		IF ((phase_horizontal_slave_position > (csp_case_feed_shuttle_horizontal.axis.actual_position + 5))
			OR
			(phase_horizontal_slave_position < (csp_case_feed_shuttle_horizontal.axis.actual_position - 5)))
		THEN
			large_move_required := TRUE;	// shuttle is moving a large amount, spreader need to be moved
		ELSE
			large_move_required := FALSE; // shuttle is moving a small amount, spreaders do not need to be moved
		END_IF
		
		IF (ABSENT_HOR_VER = FALSE) 
			AND (csp_case_flapControl.spreaders_clear
			OR
			large_move_required = FALSE)
		THEN
			axis_move_absolute(
				position 		:= phase_horizontal_slave_position,
				velocity 		:= csp_case_feed_shuttle_horizontal.MOTOR_PHASE_VELOCITY_MMPS,
				direction		:= AXIS_CURRENT_DIRECTION,
				acceleration 	:= csp_case_feed_shuttle_horizontal.MOTOR_MAX_ACCELLERATION_MMPS2,
				deceleration 	:= csp_case_feed_shuttle_horizontal.MOTOR_MAX_DECELLERATION_MMPS2, 
				jerk 			:=csp_case_feed_shuttle_horizontal. MOTOR_MAX_JERK_MMPS3, 
				buffer_mode 	:= AXIS_BUFFER_MODE_BUFFERED,
				CONVERSION_this := csp_case_feed_shuttle_horizontal.axis); 
	
			axis_move_absolute(
				position 		:= phase_vertical_slave_position,
				velocity 		:= csp_case_feed_shuttle_vertical.MOTOR_PHASE_VELOCITY_DEGPS,
				direction		:= AXIS_SHORTEST_WAY,
				acceleration 	:= csp_case_feed_shuttle_vertical.MOTOR_MAX_ACCELLERATION_DEGPS2,
				deceleration 	:= csp_case_feed_shuttle_vertical.MOTOR_MAX_DECELLERATION_DEGPS2, 
				jerk 			:= csp_case_feed_shuttle_vertical.MOTOR_MAX_JERK_DEGPS3, 
				buffer_mode 	:= AXIS_BUFFER_MODE_BUFFERED,
				CONVERSION_this := csp_case_feed_shuttle_vertical.axis); 
		END_IF
	 	
	
			axis_move_absolute(
				position 		:= phase_x_slave_position,
				velocity 		:= csp_case_feed_kinematic_x.MOTOR_PHASE_VELOCITY_MMPS,
				direction		:= AXIS_CURRENT_DIRECTION,
				acceleration 	:= csp_case_feed_kinematic_x.MOTOR_MAX_ACCELLERATION_MMPS2,
				deceleration 	:= csp_case_feed_kinematic_x.MOTOR_MAX_DECELLERATION_MMPS2, 
				jerk 			:= csp_case_feed_kinematic_x.MOTOR_MAX_JERK_MMPS3, 
				buffer_mode 	:= AXIS_BUFFER_MODE_BUFFERED,
				CONVERSION_this := csp_case_feed_kinematic_x.axis); 
			
			axis_move_absolute(
				position 		:= phase_y_slave_position,
				velocity 		:= csp_case_feed_kinematic_y.MOTOR_PHASE_VELOCITY_MMPS,
				direction		:= AXIS_CURRENT_DIRECTION,
				acceleration 	:= csp_case_feed_kinematic_y.MOTOR_MAX_ACCELLERATION_MMPS2,
				deceleration 	:= csp_case_feed_kinematic_y.MOTOR_MAX_DECELLERATION_MMPS2, 
				jerk 			:= csp_case_feed_kinematic_y.MOTOR_MAX_JERK_MMPS3, 
				buffer_mode 	:= AXIS_BUFFER_MODE_BUFFERED,
				CONVERSION_this := csp_case_feed_kinematic_y.axis); 
			
			axis_move_absolute(
				position 		:= phase_tilt_slave_position,
				velocity 		:= csp_case_feed_kinematic_tilt.MOTOR_PHASE_VELOCITY_DEGPS,
				direction		:= AXIS_CURRENT_DIRECTION,
				acceleration 	:= csp_case_feed_kinematic_tilt.MOTOR_MAX_ACCELLERATION_DEGPS2,
				deceleration 	:= csp_case_feed_kinematic_tilt.MOTOR_MAX_DECELLERATION_DEGPS2, 
				jerk 			:= csp_case_feed_kinematic_tilt.MOTOR_MAX_JERK_DEGPS3, 
				buffer_mode 	:= AXIS_BUFFER_MODE_BUFFERED,
				CONVERSION_this := csp_case_feed_kinematic_tilt.axis); 
			
		IF 	axis_is_absolute_moving(csp_case_feed_shuttle_horizontal.axis)
			AND
			axis_is_absolute_moving(csp_case_feed_shuttle_vertical.axis)
			AND
			axis_is_absolute_moving(csp_case_feed_kinematic_x.axis)
			AND
			axis_is_absolute_moving(csp_case_feed_kinematic_y.axis)
			AND
			axis_is_absolute_moving(csp_case_feed_kinematic_tilt.axis)
		THEN
			csp_case_feed_kinematic.ext_phase_request := TRUE;
			phase_status_next := CSP_CASE_FEED_STATUS_PHASE_MOVED_SLAVE_POSITION;
		ELSIF 	ABSENT_HOR_VER
				AND
				axis_is_absolute_moving(csp_case_feed_kinematic_x.axis)
				AND
				axis_is_absolute_moving(csp_case_feed_kinematic_y.axis)
				AND
				axis_is_absolute_moving(csp_case_feed_kinematic_tilt.axis)
		THEN
				csp_case_feed_kinematic.ext_phase_request := TRUE;
				phase_status_next := CSP_CASE_FEED_STATUS_PHASE_MOVED_SLAVE_POSITION;
		END_IF

		
	CSP_CASE_FEED_STATUS_PHASE_MOVED_SLAVE_POSITION:
	
		IF 	((axis_is_standstill(csp_case_feed_shuttle_horizontal.axis)
			AND
			axis_is_standstill(csp_case_feed_shuttle_vertical.axis))
			OR
			ABSENT_HOR_VER)
			AND
			axis_is_standstill(csp_case_feed_kinematic_x.axis)
			AND
			axis_is_standstill(csp_case_feed_kinematic_y.axis)
			AND
			axis_is_standstill(csp_case_feed_kinematic_tilt.axis)
			AND
			csp_case_feed_kinematic.phase_request
		THEN			
			phase_status_next := CSP_CASE_FEED_STATUS_PHASE_DONE;
		END_IF
					
		
	CSP_CASE_FEED_STATUS_PHASE_DONE:	(* Phase done *)
			
		phase_running := FALSE;
		phase_done := TRUE;			

		IF 	csp_case_feed_kinematic.ext_stop_request	
		THEN
			phase_done := FALSE;
			phase_status_next := CSP_CASE_FEED_STATUS_PHASE_START;
		END_IF
		
		
	CSP_CASE_FEED_STATUS_PHASE_ERROR:	(* Phase error *)
	
		IF	phase_running
		THEN
			axis_disable(csp_case_feed_shuttle_horizontal.axis);
			axis_disable(csp_case_feed_shuttle_vertical.axis);									
		END_IF
		phase_running := FALSE;
		
		IF	phase_conditions 	
		THEN
			phase_status_next := CSP_CASE_FEED_STATUS_PHASE_START;
		END_IF
		
END_CASE

IF 	NOT debug_state_machine
	OR
	debug_phase_machine_one_step	
THEN
	phase_status := phase_status_next;
	debug_phase_machine_one_step := FALSE;
END_IF

(* Phasing timeout *)
IF	phase_running
	AND NOT debug_state_machine
THEN
	IF	timer_is_expired(phase_time_out_tmr)
	THEN
		process_message_set(1, phase_status, 0, phase_faulted_aem);
	END_IF
ELSE
	timer_restart(30000, phase_time_out_tmr);
END_IF
END_ACTION

END_PROGRAM

// ---- POUs/AFL extensions/jog_manager/status/jog_manager_is_jog_axis_active.TcPOU
(*$
	Returns <i>TRUE</i> if the status of the instance <b><i>this</i></b> is
	<a href="#jog_manager_status_enum"><i>JOG_MANAGER_STATUS_ACTIVE</i></a>
	and  <i>list_selected</i> is a valid index,
	<i>FALSE</i> otherwise.
$*)
FUNCTION jog_manager_is_jog_axis_active : BOOL
VAR_INPUT
	index:				UINT;
END_VAR
VAR_IN_OUT
    CONVERSION_this:	jog_manager;	(*$ Instance to which the method applies $*)
END_VAR

IF	(
		(CONVERSION_this.CONVERSION_private.list_selected = index)
		OR 	
		(CONVERSION_this.CONVERSION_private.old_list_selected = index)
	)
	AND
	CONVERSION_this.CONVERSION_private.list_selected_axis_is_valid
THEN
	jog_manager_is_jog_axis_active := (CONVERSION_this.status >= JOG_MANAGER_STATUS_ACTIVE);
ELSE
	jog_manager_is_jog_axis_active := FALSE;
END_IF

END_FUNCTION

// ---- Application/CSP/Case/Feed/Kinematic/csp_case_feed_kinematic.TcPOU
(*********************************** G.D S.p.A. - Technical Department ***********************************
============= PROGRAM INFO ============
FOLDER:             TBD
MACHINES INVOLVED:  TBD 

============= DESCRIPTION =============
csp machine declaration

============= REVISIONS ===============
Date		Version	 	Author      	Description             
----------	-------		------------  	--------------------------------------------
2019/04/05 	0000.00	 	M.Grasso		Creation of the PRG

**********************************************************************************************************)
(*$R process_ref := prc; $*)
PROGRAM csp_case_feed_kinematic
VAR_INPUT
	ext_cartesian_mode_request:						BOOL;
	ext_phase_request:								BOOL;
	ext_stop_request:								BOOL;
END_VAR
VAR
	
	prc:											process;
	prc_path:										STRING;
	
	in_stKinToPlc	AT %I*:							NcToPlc_NciChannel_Ref;
	out_stPlcToKin	AT %Q*:							PlcTonc_NciChannel_Ref;
	stAxesConfig:									ST_KinAxes;
	stAxesPosIn:									ARRAY[1..8] OF LREAL;
	stAxesPosOut:									ARRAY[1..8] OF LREAL;
	uMetaInfoIn:									U_KinMetaInfo;
	uMetaInfoOut:									U_KinMetaInfo;
		
	kin_config_execute:								BOOL := FALSE;
	kin_config_cartesian_mode:						BOOL := FALSE;
	fbConfigKinGroup:								FB_KinConfigGroup;
	kin_config_group_aem:	 						message;	
	kin_cacl_execute:								BOOL := FALSE;
	fbCalcKinTrafo:									FB_KinCalcTRafo;
	fbResetKinGroup:								FB_KinResetGroup;
	
	fsm_enable_condition:							BOOL := FALSE;
	fsm_next_status:								csp_case_feed_kinematic_status_enum;
	fsm_status:										csp_case_feed_kinematic_status_enum;
			
	kinematic_jog_on:								BOOL := FALSE; (*$P $*)
	kinematic_jog_on_motcond:						motorization_conditioner;
	
	memo_cartesian_mode_request:					BOOL;
	memo_phase_request:								BOOL;
	memo_stop_request:								BOOL;
	
	cartesian_mode_active:							BOOL;
	is_ok:											BOOL;
	is_axis_enabled:								BOOL;
	
	disable_req:									BOOL := FALSE;
	move_kinematic:									BOOL := TRUE;
	enable_kinematic:								BOOL := TRUE;
	engage_enable:									BOOL := FALSE;
	disable_kinematic:								BOOL := TRUE;
	
	//Cmd	
	joint_cartesian_mode:							BOOL := FALSE;
	join_cartesian_mode_RTRIG:						R_TRIG;
	
	elbow_jog_plus:									BOOL := FALSE;
	elbow_jog_minus:								BOOL := FALSE;
	elbow_phase_move:								BOOL := FALSE;
	elbow_copy_phase:								BOOL := FALSE;
	
	shoulder_jog_plus:								BOOL := FALSE;
	shoulder_jog_minus:								BOOL := FALSE;
	shoulder_phase_move:							BOOL := FALSE;
	shoulder_copy_phase:							BOOL := FALSE;
	
	wrist_jog_plus:									BOOL := FALSE;
	wrist_jog_minus:								BOOL := FALSE;
	wrist_phase_move:								BOOL := FALSE;	
	wrist_copy_phase:								BOOL := FALSE;	

	x_jog_plus:										BOOL := FALSE;
	x_jog_minus:									BOOL := FALSE;
	x_phase_move:									BOOL := FALSE;
	x_copy_phase:									BOOL := FALSE;
	
	y_jog_plus:										BOOL := FALSE;
	y_jog_minus:									BOOL := FALSE;
	y_phase_move:									BOOL := FALSE;
	y_copy_phase:									BOOL := FALSE;
	
	tilt_jog_plus:									BOOL := FALSE;
	tilt_jog_minus:									BOOL := FALSE;
	tilt_phase_move:								BOOL := FALSE;	
	tilt_copy_phase:								BOOL := FALSE;
	
	elbow_move_speed:								LREAL := 5.0; 		(*$P unit := °/s; $*)
	shoulder_move_speed:							LREAL := 5.0;		(*$P unit := °/s; $*)
	wrist_move_speed:								LREAL := 5.0;		(*$P unit := °/s; $*)
	x_move_speed:									LREAL := 10.0;		(*$P unit := mm/s; $*)
	y_move_speed:									LREAL := 10.0;		(*$P unit := mm/s; $*)
	tilt_move_speed:								LREAL := 10.0;		(*$P unit := °/s; $*)
	
	phase_move_speed:								LREAL := 10;
	phase_move_time:								LREAL;
	x_phase_distance:								LREAL;
	x_phase_move_speed:								LREAL;
	y_phase_distance:								LREAL;	
	y_phase_move_speed:								LREAL;	
		
	phase_request:									BOOL := FALSE;
	elbow_phase_position:							LREAL := 0.0;		(*$P step := 0.001; unit := °; $*)
	elbow_phase_position_pow:						parameter_overwrite;
	shoulder_phase_position:						LREAL := 45.0;		(*$P step := 0.001; unit := °; $*)
	shoulder_phase_position_pow:					parameter_overwrite;
	wrist_phase_position:							LREAL := 0.0;		(*$P step := 0.001; unit := °; $*)
	wrist_phase_position_pow:						parameter_overwrite;
	x_phase_position:								LREAL := -554;		(*$P step := 0.001; unit := mm; $*)
	x_phase_position_pow:							parameter_overwrite;
	y_phase_position:								LREAL := -660.3;	(*$P step := 0.001; unit := mm; $*)
	y_phase_position_pow:							parameter_overwrite;
	tilt_phase_position:							LREAL := 45.0;		(*$P step := 0.001; unit := °; $*)
	tilt_phase_position_pow:						parameter_overwrite;
	
	elbow_actual_position:							LREAL;				(*$M step := 0.001; unit := °; $*)
	shoulder_actual_position:						LREAL;				(*$M step := 0.001; unit := °; $*)
	wrist_actual_position:							LREAL;				(*$M step := 0.001; unit := °; $*)
	x_actual_position:								LREAL;				(*$M step := 0.01; unit := mm; $*)
	y_actual_position:								LREAL;				(*$M step := 0.01; unit := mm; $*)
	tilt_actual_position:							LREAL;				(*$M step := 0.01; unit := °; $*)
	axis_are_moving:								BOOL;
	axis_are_phase_moving:							BOOL;
	
	//Visu variable management	
	visu_disable_general_command:					BOOL;
	visu_disable_ACS_command:						BOOL;
	visu_disable_MCS_command:						BOOL;
	visu_disable_ACS_jog_mode:						BOOL;
	visu_disable_MCS_jog_mode:						BOOL;
	visu_disable_phase_request:						BOOL;
	
	//HMI custom page variable management
	hmi_joint_cartesian_mode_cbtn:					command_button;
	hmi_phase_request_cbtn:							command_button;
	hmi_phase_request_cbtn_is_pressed:				BOOL;	
	
	hmi_elbow_jog_plus_cbtn:						command_button;
	hmi_elbow_jog_minus_cbtn:						command_button;
	hmi_elbow_phase_move_cbtn:						command_button;
	hmi_elbow_copy_phase_cbtn:						command_button;
	hmi_elbow_activate_pendant_cbtn:				command_button;
	hmi_elbow_activate_pendant_cbtn_is_pressed:		BOOL;
	hmi_elbow_pendant_active:						BOOL := FALSE;
	
	hmi_shoulder_jog_plus_cbtn:						command_button;
	hmi_shoulder_jog_minus_cbtn:					command_button;
	hmi_shoulder_phase_move_cbtn:					command_button;
	hmi_shoulder_copy_phase_cbtn:					command_button;
	hmi_shoulder_activate_pendant_cbtn:				command_button;
	hmi_shoulder_activate_pendant_cbtn_is_pressed:	BOOL;
	hmi_shoulder_pendant_active:					BOOL := FALSE;
	
	hmi_wrist_jog_plus_cbtn:						command_button;
	hmi_wrist_jog_minus_cbtn:						command_button;
	hmi_wrist_phase_move_cbtn:						command_button;
	hmi_wrist_copy_phase_cbtn:						command_button;
	hmi_wrist_activate_pendant_cbtn:				command_button;
	hmi_wrist_activate_pendant_cbtn_is_pressed:		BOOL;
	hmi_wrist_pendant_active:						BOOL := FALSE;
	
	hmi_x_jog_plus_cbtn:							command_button;
	hmi_x_jog_minus_cbtn:							command_button;
	hmi_x_phase_move_cbtn:							command_button;
	hmi_x_copy_phase_cbtn:							command_button;
	hmi_x_activate_pendant_cbtn:					command_button;
	hmi_x_activate_pendant_cbtn_is_pressed:			BOOL;
	hmi_x_pendant_active:							BOOL := FALSE;
	
	hmi_y_jog_plus_cbtn:							command_button;
	hmi_y_jog_minus_cbtn:							command_button;
	hmi_y_phase_move_cbtn:							command_button;
	hmi_y_copy_phase_cbtn:							command_button;
	hmi_y_activate_pendant_cbtn:					command_button;
	hmi_y_activate_pendant_cbtn_is_pressed:			BOOL;
	hmi_y_pendant_active:							BOOL := FALSE;
	
	hmi_tilt_jog_plus_cbtn:							command_button;
	hmi_tilt_jog_minus_cbtn:						command_button;
	hmi_tilt_phase_move_cbtn:						command_button;
	hmi_tilt_copy_phase_cbtn:						command_button;
	hmi_tilt_activate_pendant_cbtn:					command_button;
	hmi_tilt_activate_pendant_cbtn_is_pressed:		BOOL;
	hmi_tilt_pendant_active:						BOOL := FALSE;
	
	hmi_pendant_active:								BOOL;
	
	hmi_enable_general_command_hgos:				hmi_graphic_object_status;
	hmi_enable_joint_hgos:							hmi_graphic_object_status;
	hmi_enable_cartesian_hgos:						hmi_graphic_object_status;
	hmi_enable_ACS_command_hgos:					hmi_graphic_object_status;
	hmi_enable_MCS_command_hgos:					hmi_graphic_object_status;
	hmi_enable_ACS_jog_mode_hgos:					hmi_graphic_object_status;
	hmi_enable_MCS_jog_mode_hgos:					hmi_graphic_object_status;
	hmi_enable_phase_request_hgos:					hmi_graphic_object_status;
	
	debug_phase_elbow:								BOOL := FALSE;
	debug_phase_shoulder:							BOOL := FALSE;
	debug_phase_wrist:								BOOL := FALSE;
	debug_state_machine:							BOOL := FALSE;
	debug_state_machine_one_step:					BOOL := FALSE;
	
	master_scaling_deg:								LREAL := 1.0;
	x_scaling_mm:									LREAL := 1.0;
	x_old_scaling_mm:								LREAL := 1.0;
	y_scaling_mm:									LREAL := 1.0;
	y_old_scaling_mm:								LREAL := 1.0;
	tilt_scaling_deg:								LREAL := 1.0;
	tilt_old_scaling_deg:							LREAL := 1.0;		
	Kinematic_tilt_error_aem: 						message;
	Kinematic_tilt_clear_error:						BOOL:= FALSE;
END_VAR

VAR CONSTANT	
	CONSTANTS:										csp_case_feed_kinematic_constant_struct;
	COIDTRAFO:										UDINT := 16#01010030;
END_VAR

_read_var_input();

_object_manager();

IF NOT objects_running()
THEN
	RETURN;	
END_IF

_read_process_image();

_mode_manager();

CASE process_get_mode(prc) of
	MODE_ABSENT,
	MODE_INACTIVE:
		RETURN;
	MODE_TEST:
		_handle_process_test();
END_CASE

_set_runtime_properties();

_hmi_Management();

(********************************* BODY *********************************)
(* Kinematic trasformation		
X		->		Shoulder (M1)
Y		->		Elbow (M2)			
Tilt	->		Wrist (M3)																											
*)	

stAxesConfig.nAxisIdsAcs[1] := csp_case_feed_arm_shoulder.axis.ax_ref.NcToPlc.AxisId; 
stAxesConfig.nAxisIdsAcs[2] := csp_case_feed_arm_elbow.axis.ax_ref.NcToPlc.AxisId;
stAxesConfig.nAxisIdsAcs[3] := csp_case_feed_arm_wrist.axis.ax_ref.NcToPlc.AxisId;

stAxesConfig.nAxisIdsMcs[1] := csp_case_feed_kinematic_x.axis.ax_ref.NcToPlc.AxisId;
stAxesConfig.nAxisIdsMcs[2] := csp_case_feed_kinematic_y.axis.ax_ref.NcToPlc.AxisId;
stAxesConfig.nAxisIdsMcs[3] := csp_case_feed_kinematic_tilt.axis.ax_ref.NcToPlc.AxisId;

fbConfigKinGroup(
	bExecute		:= kin_config_execute
					   OR
					   (
						   (
							   NOT axis_is_ok(FALSE, csp_case_feed_arm_elbow.axis)
							   OR
							   NOT axis_is_ok(FALSE, csp_case_feed_arm_shoulder.axis)
							   OR
							   NOT axis_is_ok(FALSE, csp_case_feed_arm_wrist.axis)	
							   OR
							   fbConfigKinGroup.bError
							)
							AND
 							csp_main.o_reset_button
					   ),
	bCartesianMode	:= kin_config_cartesian_mode, 
	stAxesList		:= stAxesConfig, 
	stKinRefIn		:= in_stKinToPlc, 
	bBusy			=> , 
	bDone			=> , 
	bError			=> , 
	nErrorId		=> );
	
fbResetKinGroup(
	bExecute		:= csp_main.o_reset_button
					AND 
					(in_stKinToPlc.ErrorCode <> 0), 
	nItpChannelId	:= 0, 
	stKinRefIn		:= in_stKinToPlc, 
	stAxesList		:= stAxesConfig, 
	bBusy			=> , 
	bDone			=> , 
	bError			=> , 
	nErrorId		=> );
	
kin_cacl_execute :=	NOT cartesian_mode_active
					AND
					NOT fbCalcKinTrafo.bBusy;
stAxesPosIn[1] := axis_get_actual_incremental_position(csp_case_feed_arm_shoulder.axis);
stAxesPosIn[2] := axis_get_actual_incremental_position(csp_case_feed_arm_elbow.axis);
stAxesPosIn[3] := axis_get_actual_incremental_position(csp_case_feed_arm_wrist.axis);
fbCalcKinTrafo(
	bExecute 		:= kin_cacl_execute,
	bForward 		:= NOT kin_config_cartesian_mode,
	oidTrafo 		:= COIDTRAFO,
	stAxesPosIn 	:= stAxesPosIn,
	stAxesPosOut 	:= stAxesPosOut,
	uMetaInfoIn		:= uMetaInfoIn ,
	uMetaInfoOut	:= uMetaInfoOut,
	bBusy			=> ,
	bDone			=> ,
	bError			=> ,
	nErrorId		=> );

(*Status*)
cartesian_mode_active := 
	(in_stKinToPlc.ChnOperationState = 4);
	
is_axis_enabled := (fsm_status = CSP_CASE_FEED_KINEMATIC_STATUS_ENABLED);
	

(* ALLOWS MACHINE TO RUN BECAUSE KINEMATIC IS NOT ON *)
IF motorization_manager_is_starting(csp_main_motorization_manager.motm)
AND NOT kinematic_jog_on
	THEN
		motorization_conditioner_start_done(kinematic_jog_on_motcond);
END_IF 


(*FSM Control*)
is_ok := 
	process_is_ready(prc)
	AND
	process_subtree_is_ready(prc)
	AND
	csp_case_feed_arm_elbow.servo_on_condition
	AND
	csp_case_feed_arm_shoulder.servo_on_condition
	AND
	csp_case_feed_arm_wrist.servo_on_condition
	AND
	axis_is_ok(FALSE, csp_case_feed_arm_elbow.axis)
	AND
	axis_is_ok(FALSE, csp_case_feed_arm_shoulder.axis)
	AND
	axis_is_ok(FALSE, csp_case_feed_arm_wrist.axis)						
	AND						
	axis_is_ok(FALSE, csp_case_feed_kinematic_x.axis)	
	AND
	axis_is_ok(FALSE, csp_case_feed_kinematic_y.axis)	
	AND
	axis_is_ok(FALSE, csp_case_feed_kinematic_tilt.axis)	
	AND												
	NOT fbConfigKinGroup.bError						
	AND
	NOT disable_req;
fsm_enable_condition := 
	is_ok
	AND
	(
		csp_case_feed_virtualMaster.is_ok
		OR
		(
			csp_main_accuChange.machine_size_running
			AND
			(
				NOT csp_case_feed_kinematic_x.in_accu_safe_pos
				OR
				NOT csp_case_feed_kinematic_y.in_accu_safe_pos
				OR
				NOT csp_case_feed_kinematic_tilt.in_accu_safe_pos
			)
		)
	);
	
IF	(
		NOT fsm_enable_condition
		OR
		(
			ext_stop_request 
			AND 
			NOT memo_stop_request
		)
	)
	AND
	fsm_status <> CSP_CASE_FEED_KINEMATIC_STATUS_DISABLED
	AND
	fsm_status < CSP_CASE_FEED_KINEMATIC_STATUS_STOP_REQUEST
THEN
	fsm_status	:=	CSP_CASE_FEED_KINEMATIC_STATUS_DISABLE_REQUEST;
	IF	ext_stop_request
	THEN
		fsm_next_status := fsm_status;
	END_IF
	phase_request:=FALSE;
END_IF

IF tilt_actual_position < 1200
	AND tilt_actual_position > 0
	AND csp_case_feed_kinematic_tilt.axis.actual_position < 1200   
	AND NOT Kinematic_tilt_clear_error
THEN
	process_message_set(1, 1, 1, Kinematic_tilt_error_aem);
ELSE
	process_message_reset(Kinematic_tilt_error_aem);
END_IF

IF process_message_is_on(Kinematic_tilt_error_aem)
	AND machine_is_stopped(csp.mch)
	OR machine_is_stop_emergency_active(csp.mch)
THEN
	process_message_reset(Kinematic_tilt_error_aem);
END_IF

CASE fsm_status OF
	
	CSP_CASE_FEED_KINEMATIC_STATUS_NOT_INITIALIZED:
	
        IF	axis_is_ok(return_when_absent := FALSE, CONVERSION_this := csp_case_feed_arm_elbow.axis)
			AND
			axis_is_ok(return_when_absent := FALSE, CONVERSION_this := csp_case_feed_arm_shoulder.axis)
			AND
			axis_is_ok(return_when_absent := FALSE, CONVERSION_this := csp_case_feed_arm_wrist.axis)
			AND
			axis_is_ok(return_when_absent := FALSE, CONVERSION_this := csp_case_feed_kinematic_x.axis)
			AND
			axis_is_ok(return_when_absent := FALSE, CONVERSION_this := csp_case_feed_kinematic_y.axis)
			AND
			axis_is_ok(return_when_absent := FALSE, CONVERSION_this := csp_case_feed_kinematic_tilt.axis)
        THEN
            fsm_next_status := CSP_CASE_FEED_KINEMATIC_STATUS_DISABLED;
        END_IF

		
	CSP_CASE_FEED_KINEMATIC_STATUS_DISABLED:
		
		IF	fsm_enable_condition
			AND (
					kinematic_jog_on
					OR
					motorization_manager_is_starting(csp_main_motorization_manager.motm)
				)
		THEN			
			fsm_next_status := CSP_CASE_FEED_KINEMATIC_STATUS_ENABLE_REQUEST;
		END_IF;

		
	CSP_CASE_FEED_KINEMATIC_STATUS_ENABLE_REQUEST:
	
		axis_enable(csp_case_feed_arm_elbow.axis);
		axis_enable(csp_case_feed_arm_shoulder.axis);
		axis_enable(csp_case_feed_arm_wrist.axis);
		axis_enable(csp_case_feed_kinematic_x.axis);
		axis_enable(csp_case_feed_kinematic_y.axis);
		axis_enable(csp_case_feed_kinematic_tilt.axis);
		
		IF 	axis_is_standstill(csp_case_feed_arm_elbow.axis)
			AND
			axis_is_standstill(csp_case_feed_arm_shoulder.axis)
			AND
			axis_is_standstill(csp_case_feed_arm_wrist.axis)
			AND
			axis_is_standstill(csp_case_feed_kinematic_x.axis)
			AND
			axis_is_standstill(csp_case_feed_kinematic_y.axis)
			AND
			axis_is_standstill(csp_case_feed_kinematic_tilt.axis)
		THEN			
			IF NOT kin_config_cartesian_mode
			   AND csp_main_accuChange.Brand_Change_Occurred
			THEN
				join_cartesian_mode_RTRIG(CLK:=FALSE);							
			END_IF
		
			fsm_next_status	:= CSP_CASE_FEED_KINEMATIC_STATUS_ENABLED;				
		END_IF;		
		
		
	CSP_CASE_FEED_KINEMATIC_STATUS_ENABLED:
	
		axis_are_phase_moving := FALSE;
		join_cartesian_mode_RTRIG(CLK := 
			joint_cartesian_mode
			OR
			command_button_is_pressed(hmi_joint_cartesian_mode_cbtn)
			OR
			csp_main_accuChange.Brand_Change_Occurred);
			
		IF	join_cartesian_mode_RTRIG.Q
		THEN
			kin_config_execute := TRUE;
			kin_config_cartesian_mode := NOT kin_config_cartesian_mode;
			fsm_next_status	:= CSP_CASE_FEED_KINEMATIC_STATUS_KIN_CONFIG;	
		ELSIF ext_cartesian_mode_request
			AND
			NOT memo_cartesian_mode_request
		THEN
			kin_config_execute := TRUE;
			kin_config_cartesian_mode := TRUE;
			fsm_next_status	:= CSP_CASE_FEED_KINEMATIC_STATUS_KIN_CONFIG;							
		ELSIF phase_request
		THEN
			IF 	motorization_manager_is_idle(csp_main_motorization_manager.motm)
			THEN			
				IF 	move_kinematic
				THEN
					fsm_next_status	:= CSP_CASE_FEED_KINEMATIC_STATUS_PHASED;
				ELSE
					fsm_next_status	:= CSP_CASE_FEED_KINEMATIC_STATUS_PHASE_REQUEST;
				END_IF
			ELSE
				phase_request := FALSE;
			END_IF	
		ELSIF ext_phase_request
			AND
			NOT memo_phase_request
		THEN
			phase_request := TRUE;	
			fsm_next_status	:= CSP_CASE_FEED_KINEMATIC_STATUS_READY_TO_ENGAGE;		
		ELSIF elbow_jog_plus
			OR
			command_button_is_pressed(hmi_elbow_jog_plus_cbtn)
			OR
			(
				hmi_elbow_pendant_active
				AND
				csp_main_jogManager.pendant_positive_cmd
			)
		THEN
			axis_move_velocity(
				velocity		:= elbow_move_speed,
				acceleration	:= CONSTANTS.MAX_ACCELERATION_MMpSEC2,
				deceleration	:= CONSTANTS.MAX_DECELERATION_MMpSEC2,
				jerk			:= CONSTANTS.MAX_JERK_MMpSEC3,
				buffer_mode		:= AXIS_BUFFER_MODE_BUFFERED,
				CONVERSION_this	:= csp_case_feed_arm_elbow.axis);
			fsm_next_status	:= CSP_CASE_FEED_KINEMATIC_STATUS_JOG_ACS1;
		ELSIF elbow_jog_minus
			OR
			command_button_is_pressed(hmi_elbow_jog_minus_cbtn)
			OR
			(
				hmi_elbow_pendant_active
				AND
				csp_main_jogManager.pendant_negative_cmd
			)
		THEN
			axis_move_velocity(
				velocity		:= -elbow_move_speed,
				acceleration	:= CONSTANTS.MAX_ACCELERATION_MMpSEC2,
				deceleration	:= CONSTANTS.MAX_DECELERATION_MMpSEC2,
				jerk			:= CONSTANTS.MAX_JERK_MMpSEC3,
				buffer_mode		:= AXIS_BUFFER_MODE_BUFFERED,
				CONVERSION_this	:= csp_case_feed_arm_elbow.axis);
			fsm_next_status	:= CSP_CASE_FEED_KINEMATIC_STATUS_JOG_ACS1;
		ELSIF elbow_phase_move
			OR
			command_button_is_pressed(hmi_elbow_phase_move_cbtn)
			OR
			debug_phase_elbow
		THEN
			debug_phase_elbow := FALSE;
			axis_are_phase_moving := TRUE;
			fsm_next_status	:= CSP_CASE_FEED_KINEMATIC_STATUS_MOVE_ACS1;			 
		ELSIF elbow_copy_phase
			OR
			command_button_is_pressed(hmi_elbow_copy_phase_cbtn)
		THEN		
			parameter_overwrite_set_lreal_value(elbow_actual_position, elbow_phase_position_pow);			
		ELSIF shoulder_jog_plus
			OR
			command_button_is_pressed(hmi_shoulder_jog_plus_cbtn)
			OR
			(
				hmi_shoulder_pendant_active
				AND
				csp_main_jogManager.pendant_positive_cmd
			)
		THEN
			axis_move_velocity(
				velocity		:= shoulder_move_speed,
				acceleration	:= CONSTANTS.MAX_ACCELERATION_MMpSEC2,
				deceleration	:= CONSTANTS.MAX_DECELERATION_MMpSEC2,
				jerk			:= CONSTANTS.MAX_JERK_MMpSEC3,
				buffer_mode		:= AXIS_BUFFER_MODE_BUFFERED,
				CONVERSION_this	:= csp_case_feed_arm_shoulder.axis);
			fsm_next_status	:= CSP_CASE_FEED_KINEMATIC_STATUS_JOG_ACS2;
		ELSIF shoulder_jog_minus
			OR
			command_button_is_pressed(hmi_shoulder_jog_minus_cbtn)
			OR
			(
				hmi_shoulder_pendant_active
				AND
				csp_main_jogManager.pendant_negative_cmd
			)
		THEN
			axis_move_velocity(
				velocity		:= -shoulder_move_speed,
				acceleration	:= CONSTANTS.MAX_ACCELERATION_MMpSEC2,
				deceleration	:= CONSTANTS.MAX_DECELERATION_MMpSEC2,
				jerk			:= CONSTANTS.MAX_JERK_MMpSEC3,
				buffer_mode		:= AXIS_BUFFER_MODE_BUFFERED,
				CONVERSION_this	:= csp_case_feed_arm_shoulder.axis);
			fsm_next_status	:= CSP_CASE_FEED_KINEMATIC_STATUS_JOG_ACS2;
		ELSIF shoulder_phase_move 
			OR
			command_button_is_pressed(hmi_shoulder_phase_move_cbtn)
			OR
			debug_phase_shoulder
		THEN
			debug_phase_shoulder := FALSE;
			axis_are_phase_moving := TRUE;
			fsm_next_status	:= CSP_CASE_FEED_KINEMATIC_STATUS_MOVE_ACS2;	
		ELSIF shoulder_copy_phase
			OR
			command_button_is_pressed(hmi_shoulder_copy_phase_cbtn)
		THEN
			parameter_overwrite_set_lreal_value(shoulder_actual_position, shoulder_phase_position_pow);							
		ELSIF wrist_jog_plus
			OR
			command_button_is_pressed(hmi_wrist_jog_plus_cbtn)
			OR
			(
				hmi_wrist_pendant_active
				AND
				csp_main_jogManager.pendant_positive_cmd
			)
		THEN
			axis_move_velocity(
				velocity		:= wrist_move_speed,
				acceleration	:= CONSTANTS.MAX_ACCELERATION_MMpSEC2,
				deceleration	:= CONSTANTS.MAX_DECELERATION_MMpSEC2,
				jerk			:= CONSTANTS.MAX_JERK_MMpSEC3,
				buffer_mode		:= AXIS_BUFFER_MODE_BUFFERED,
				CONVERSION_this	:= csp_case_feed_arm_wrist.axis);
			fsm_next_status	:= CSP_CASE_FEED_KINEMATIC_STATUS_JOG_ACS3;
		ELSIF wrist_jog_minus
			OR
			command_button_is_pressed(hmi_wrist_jog_minus_cbtn)
			OR
			(
				hmi_wrist_pendant_active
				AND
				csp_main_jogManager.pendant_negative_cmd
			)
		THEN
			axis_move_velocity(
				velocity		:= -wrist_move_speed,
				acceleration	:= CONSTANTS.MAX_ACCELERATION_MMpSEC2,
				deceleration	:= CONSTANTS.MAX_DECELERATION_MMpSEC2,
				jerk			:= CONSTANTS.MAX_JERK_MMpSEC3,
				buffer_mode		:= AXIS_BUFFER_MODE_BUFFERED,
				CONVERSION_this	:= csp_case_feed_arm_wrist.axis);
			fsm_next_status	:= CSP_CASE_FEED_KINEMATIC_STATUS_JOG_ACS3;
		ELSIF wrist_phase_move
			OR
			command_button_is_pressed(hmi_wrist_phase_move_cbtn)
			OR
			debug_phase_wrist
		THEN
			debug_phase_wrist := FALSE;
			axis_are_phase_moving := TRUE;
			fsm_next_status	:= CSP_CASE_FEED_KINEMATIC_STATUS_MOVE_ACS3;
		ELSIF wrist_copy_phase
			OR
			command_button_is_pressed(hmi_wrist_copy_phase_cbtn)
		THEN			
			parameter_overwrite_set_lreal_value(wrist_actual_position, wrist_phase_position_pow);			
		ELSIF x_jog_plus
			OR
			command_button_is_pressed(hmi_x_jog_plus_cbtn)
			OR
			(
				hmi_x_pendant_active
				AND
				csp_main_jogManager.pendant_positive_cmd
			)
		THEN
			axis_move_velocity(
				velocity		:= x_move_speed,
				acceleration	:= CONSTANTS.MAX_ACCELERATION_MMpSEC2,
				deceleration	:= CONSTANTS.MAX_DECELERATION_MMpSEC2,
				jerk			:= CONSTANTS.MAX_JERK_MMpSEC3,
				buffer_mode		:= AXIS_BUFFER_MODE_BUFFERED,
				CONVERSION_this	:= csp_case_feed_kinematic_x.axis);
			fsm_next_status	:= CSP_CASE_FEED_KINEMATIC_STATUS_JOG_MCS1;						
		ELSIF x_jog_minus
			OR
			command_button_is_pressed(hmi_x_jog_minus_cbtn)
			OR
			(
				hmi_x_pendant_active
				AND
				csp_main_jogManager.pendant_negative_cmd
			)
		THEN
			axis_move_velocity(
				velocity		:= -x_move_speed,
				acceleration	:= CONSTANTS.MAX_ACCELERATION_MMpSEC2,
				deceleration	:= CONSTANTS.MAX_DECELERATION_MMpSEC2,
				jerk			:= CONSTANTS.MAX_JERK_MMpSEC3,
				buffer_mode		:= AXIS_BUFFER_MODE_BUFFERED,
				CONVERSION_this	:= csp_case_feed_kinematic_x.axis);
			fsm_next_status	:= CSP_CASE_FEED_KINEMATIC_STATUS_JOG_MCS1;
		ELSIF x_phase_move
			OR
			command_button_is_pressed(hmi_x_phase_move_cbtn)
		THEN
			axis_are_phase_moving := TRUE;
			fsm_next_status	:= CSP_CASE_FEED_KINEMATIC_STATUS_MOVE_MCS1;
		ELSIF x_copy_phase
			OR
			command_button_is_pressed(hmi_x_copy_phase_cbtn)
		THEN			
			parameter_overwrite_set_lreal_value(x_actual_position, x_phase_position_pow);			
		ELSIF y_jog_plus
			OR
			command_button_is_pressed(hmi_y_jog_plus_cbtn)
			OR
			(
				hmi_y_pendant_active
				AND
				csp_main_jogManager.pendant_positive_cmd
			)
		THEN
			axis_move_velocity(
				velocity		:= y_move_speed,
				acceleration	:= CONSTANTS.MAX_ACCELERATION_MMpSEC2,
				deceleration	:= CONSTANTS.MAX_DECELERATION_MMpSEC2,
				jerk			:= CONSTANTS.MAX_JERK_MMpSEC3,
				buffer_mode		:= AXIS_BUFFER_MODE_BUFFERED,
				CONVERSION_this	:= csp_case_feed_kinematic_y.axis);
			fsm_next_status	:= CSP_CASE_FEED_KINEMATIC_STATUS_JOG_MCS2;
		ELSIF y_jog_minus
			OR
			command_button_is_pressed(hmi_y_jog_minus_cbtn)
			OR
			(
				hmi_y_pendant_active
				AND
				csp_main_jogManager.pendant_negative_cmd
			)
		THEN
			axis_move_velocity(
				velocity		:= -y_move_speed,
				acceleration	:= CONSTANTS.MAX_ACCELERATION_MMpSEC2,
				deceleration	:= CONSTANTS.MAX_DECELERATION_MMpSEC2,
				jerk			:= CONSTANTS.MAX_JERK_MMpSEC3,
				buffer_mode		:= AXIS_BUFFER_MODE_BUFFERED,
				CONVERSION_this	:= csp_case_feed_kinematic_y.axis);
			fsm_next_status	:= CSP_CASE_FEED_KINEMATIC_STATUS_JOG_MCS2;
		ELSIF y_phase_move
			OR
			command_button_is_pressed(hmi_y_phase_move_cbtn)
		THEN
			axis_are_phase_moving := TRUE;
			fsm_next_status	:= CSP_CASE_FEED_KINEMATIC_STATUS_MOVE_MCS2;		
		ELSIF y_copy_phase
			OR
			command_button_is_pressed(hmi_y_copy_phase_cbtn)
		THEN			
			parameter_overwrite_set_lreal_value(y_actual_position, y_phase_position_pow);							
		ELSIF tilt_jog_plus
			OR
			command_button_is_pressed(hmi_tilt_jog_plus_cbtn)
			OR
			(
				hmi_tilt_pendant_active
				AND
				csp_main_jogManager.pendant_positive_cmd
			)
		THEN
			axis_move_velocity(
				velocity		:= tilt_move_speed,
				acceleration	:= CONSTANTS.MAX_ACCELERATION_MMpSEC2,
				deceleration	:= CONSTANTS.MAX_DECELERATION_MMpSEC2,
				jerk			:= CONSTANTS.MAX_JERK_MMpSEC3,
				buffer_mode		:= AXIS_BUFFER_MODE_BUFFERED,
				CONVERSION_this	:= csp_case_feed_kinematic_tilt.axis);
			fsm_next_status	:= CSP_CASE_FEED_KINEMATIC_STATUS_JOG_MCS3;
		ELSIF tilt_jog_minus
			OR
			command_button_is_pressed(hmi_tilt_jog_minus_cbtn)
			OR
			(
				hmi_tilt_pendant_active
				AND
				csp_main_jogManager.pendant_negative_cmd
			)
		THEN
			axis_move_velocity(
				velocity		:= -tilt_move_speed,
				acceleration	:= CONSTANTS.MAX_ACCELERATION_MMpSEC2,
				deceleration	:= CONSTANTS.MAX_DECELERATION_MMpSEC2,
				jerk			:= CONSTANTS.MAX_JERK_MMpSEC3,
				buffer_mode		:= AXIS_BUFFER_MODE_BUFFERED,
				CONVERSION_this	:= csp_case_feed_kinematic_tilt.axis);
			fsm_next_status	:= CSP_CASE_FEED_KINEMATIC_STATUS_JOG_MCS3;
		ELSIF tilt_phase_move
			OR
			command_button_is_pressed(hmi_tilt_phase_move_cbtn)
		THEN
			axis_are_phase_moving := TRUE;
			fsm_next_status	:= CSP_CASE_FEED_KINEMATIC_STATUS_MOVE_MCS3;		
		ELSIF tilt_copy_phase
			OR
			command_button_is_pressed(hmi_tilt_copy_phase_cbtn)
		THEN			
			parameter_overwrite_set_lreal_value(tilt_actual_position, tilt_phase_position_pow);								
		END_IF
		
		
	CSP_CASE_FEED_KINEMATIC_STATUS_KIN_CONFIG:
	
		IF	fbConfigKinGroup.bDone
			OR
			fbConfigKinGroup.bError
		THEN
			move_kinematic := TRUE;	
			kin_config_execute := FALSE;
			fsm_next_status	:= CSP_CASE_FEED_KINEMATIC_STATUS_ENABLED;				
		END_IF
		
		
	CSP_CASE_FEED_KINEMATIC_STATUS_JOG_ACS1:
	
		IF	NOT elbow_jog_plus
			AND
			NOT elbow_jog_minus
			AND
			NOT command_button_is_pressed(hmi_elbow_jog_plus_cbtn)
			AND
			NOT command_button_is_pressed(hmi_elbow_jog_minus_cbtn)
			AND
			(
				NOT hmi_elbow_pendant_active
				OR
				(
					NOT csp_main_jogManager.pendant_positive_cmd
					AND
					axis_is_moving_forward(csp_case_feed_arm_elbow.axis)
				)
				OR
				(
					NOT csp_main_jogManager.pendant_negative_cmd
					AND
					axis_is_moving_backward(csp_case_feed_arm_elbow.axis)
				)
			)
		THEN
			axis_stop(
		    	deceleration 	:= CONSTANTS.MAX_DECELERATION_MMpSEC2,
		    	jerk 			:= CONSTANTS.MAX_JERK_MMpSEC3,
		    	CONVERSION_this := csp_case_feed_arm_elbow.axis);
			fsm_next_status	:= CSP_CASE_FEED_KINEMATIC_STATUS_STOP_ACS1;
		END_IF
		
		
	CSP_CASE_FEED_KINEMATIC_STATUS_MOVE_ACS1:
	
		axis_move_absolute(
			position 		:= elbow_phase_position,
			velocity 		:= elbow_move_speed,
			direction		:= AXIS_CURRENT_DIRECTION,
			acceleration 	:= CONSTANTS.MAX_ACCELERATION_MMpSEC2,
			deceleration 	:= CONSTANTS.MAX_DECELERATION_MMpSEC2,
			jerk 			:= CONSTANTS.MAX_JERK_MMpSEC3, 
			buffer_mode 	:= AXIS_BUFFER_MODE_BUFFERED,
			CONVERSION_this := csp_case_feed_arm_elbow.axis);
				
		IF	axis_is_absolute_moving(csp_case_feed_arm_elbow.axis)
		THEN
			fsm_next_status	:= CSP_CASE_FEED_KINEMATIC_STATUS_STOP_ACS1;
		END_IF
				
		
	CSP_CASE_FEED_KINEMATIC_STATUS_STOP_ACS1:
	
		IF	axis_is_standstill(csp_case_feed_arm_elbow.axis)
		THEN			
			fsm_next_status	:= CSP_CASE_FEED_KINEMATIC_STATUS_ENABLED;
		END_IF
	
		
	CSP_CASE_FEED_KINEMATIC_STATUS_JOG_ACS2:
	
		IF	NOT shoulder_jog_plus
			AND
			NOT shoulder_jog_minus
			AND
			NOT command_button_is_pressed(hmi_shoulder_jog_plus_cbtn)
			AND
			NOT command_button_is_pressed(hmi_shoulder_jog_minus_cbtn)
			AND
			(
				NOT hmi_shoulder_pendant_active
				OR
				(
					NOT csp_main_jogManager.pendant_positive_cmd
					AND
					axis_is_moving_forward(csp_case_feed_arm_shoulder.axis)
				)
				OR
				(
					NOT csp_main_jogManager.pendant_negative_cmd
					AND
					axis_is_moving_backward(csp_case_feed_arm_shoulder.axis)
				)
			)
		THEN
			axis_stop(
		    	deceleration 	:= CONSTANTS.MAX_DECELERATION_MMpSEC2,
		    	jerk 			:= CONSTANTS.MAX_JERK_MMpSEC3,
		    	CONVERSION_this := csp_case_feed_arm_shoulder.axis);
			fsm_next_status	:= CSP_CASE_FEED_KINEMATIC_STATUS_STOP_ACS2;
		END_IF
	
		
	CSP_CASE_FEED_KINEMATIC_STATUS_MOVE_ACS2:
	
		axis_move_absolute(
			position 		:= shoulder_phase_position,
			velocity 		:= shoulder_move_speed,
			direction		:= AXIS_CURRENT_DIRECTION,
			acceleration 	:= CONSTANTS.MAX_ACCELERATION_MMpSEC2,
			deceleration 	:= CONSTANTS.MAX_DECELERATION_MMpSEC2,
			jerk 			:= CONSTANTS.MAX_JERK_MMpSEC3, 
			buffer_mode 	:= AXIS_BUFFER_MODE_BUFFERED,
			CONVERSION_this := csp_case_feed_arm_shoulder.axis);
				
		IF	axis_is_absolute_moving(csp_case_feed_arm_shoulder.axis)
		THEN
			fsm_next_status	:= CSP_CASE_FEED_KINEMATIC_STATUS_STOP_ACS2;
		END_IF
	
		
	CSP_CASE_FEED_KINEMATIC_STATUS_STOP_ACS2:
	
		IF	axis_is_standstill(csp_case_feed_arm_shoulder.axis)
		THEN			
			fsm_next_status	:= CSP_CASE_FEED_KINEMATIC_STATUS_ENABLED;
		END_IF
	
		
	CSP_CASE_FEED_KINEMATIC_STATUS_JOG_ACS3:
	
		IF	NOT wrist_jog_plus
			AND
			NOT wrist_jog_minus
			AND
			NOT command_button_is_pressed(hmi_wrist_jog_plus_cbtn)
			AND
			NOT command_button_is_pressed(hmi_wrist_jog_minus_cbtn)
			AND
			(
				NOT hmi_wrist_pendant_active
				OR
				(
					NOT csp_main_jogManager.pendant_positive_cmd
					AND
					axis_is_moving_forward(csp_case_feed_arm_wrist.axis)
				)
				OR
				(
					NOT csp_main_jogManager.pendant_negative_cmd
					AND
					axis_is_moving_backward(csp_case_feed_arm_wrist.axis)
				)
			)
		THEN
			axis_stop(
		    	deceleration 	:= CONSTANTS.MAX_DECELERATION_MMpSEC2,
		    	jerk 			:= CONSTANTS.MAX_JERK_MMpSEC3,
		    	CONVERSION_this := csp_case_feed_arm_wrist.axis);
			fsm_next_status	:= CSP_CASE_FEED_KINEMATIC_STATUS_STOP_ACS3;
		END_IF
	
		
	CSP_CASE_FEED_KINEMATIC_STATUS_MOVE_ACS3:
	
		axis_move_absolute(
			position 		:= wrist_phase_position,
			velocity 		:= wrist_move_speed,
			direction		:= AXIS_CURRENT_DIRECTION,
			acceleration 	:= CONSTANTS.MAX_ACCELERATION_MMpSEC2,
			deceleration 	:= CONSTANTS.MAX_DECELERATION_MMpSEC2,
			jerk 			:= CONSTANTS.MAX_JERK_MMpSEC3, 
			buffer_mode 	:= AXIS_BUFFER_MODE_BUFFERED,
			CONVERSION_this := csp_case_feed_arm_wrist.axis);
				
		IF	axis_is_absolute_moving(csp_case_feed_arm_wrist.axis)
		THEN
			fsm_next_status	:= CSP_CASE_FEED_KINEMATIC_STATUS_STOP_ACS3;
		END_IF
	
		
	CSP_CASE_FEED_KINEMATIC_STATUS_STOP_ACS3:
	
		IF	axis_is_standstill(csp_case_feed_arm_wrist.axis)
		THEN			
			fsm_next_status	:= CSP_CASE_FEED_KINEMATIC_STATUS_ENABLED;
		END_IF
	
		
	CSP_CASE_FEED_KINEMATIC_STATUS_JOG_MCS1:
	
		IF	NOT x_jog_plus
			AND
			NOT x_jog_minus
			AND
			NOT command_button_is_pressed(hmi_x_jog_plus_cbtn)
			AND
			NOT command_button_is_pressed(hmi_x_jog_minus_cbtn)
			AND
			(
				NOT hmi_x_pendant_active
				OR
				(
					NOT csp_main_jogManager.pendant_positive_cmd
					AND
					axis_is_moving_forward(csp_case_feed_kinematic_x.axis)
				)
				OR
				(
					NOT csp_main_jogManager.pendant_negative_cmd
					AND
					axis_is_moving_backward(csp_case_feed_kinematic_x.axis)
				)
			)
		THEN
			axis_stop(
		    	deceleration 	:= CONSTANTS.MAX_DECELERATION_MMpSEC2,
		    	jerk 			:= CONSTANTS.MAX_JERK_MMpSEC3,
		    	CONVERSION_this := csp_case_feed_kinematic_x.axis);
			fsm_next_status	:= CSP_CASE_FEED_KINEMATIC_STATUS_STOP_MCS1;
		END_IF
	
		
	CSP_CASE_FEED_KINEMATIC_STATUS_MOVE_MCS1:
	
		axis_move_absolute(
			position 		:= x_phase_position,
			velocity 		:= x_move_speed,
			direction		:= AXIS_CURRENT_DIRECTION,
			acceleration 	:= CONSTANTS.MAX_ACCELERATION_MMpSEC2,
			deceleration 	:= CONSTANTS.MAX_DECELERATION_MMpSEC2,
			jerk 			:= CONSTANTS.MAX_JERK_MMpSEC3, 
			buffer_mode 	:= AXIS_BUFFER_MODE_BUFFERED,
			CONVERSION_this := csp_case_feed_kinematic_x.axis);
				
		IF	axis_is_absolute_moving(csp_case_feed_kinematic_x.axis)
		THEN
			fsm_next_status	:= CSP_CASE_FEED_KINEMATIC_STATUS_STOP_MCS1;
		END_IF
		
		
	CSP_CASE_FEED_KINEMATIC_STATUS_STOP_MCS1:
	
		IF	axis_is_standstill(csp_case_feed_kinematic_x.axis)
		THEN			
			fsm_next_status	:= CSP_CASE_FEED_KINEMATIC_STATUS_ENABLED;
		END_IF
	
		
	CSP_CASE_FEED_KINEMATIC_STATUS_JOG_MCS2:
	
		IF	NOT y_jog_plus
			AND
			NOT y_jog_minus
			AND
			NOT command_button_is_pressed(hmi_y_jog_plus_cbtn)
			AND
			NOT command_button_is_pressed(hmi_y_jog_minus_cbtn)
			AND
			(
				NOT hmi_y_pendant_active
				OR
				(
					NOT csp_main_jogManager.pendant_positive_cmd
					AND
					axis_is_moving_forward(csp_case_feed_kinematic_y.axis)
				)
				OR
				(
					NOT csp_main_jogManager.pendant_negative_cmd
					AND
					axis_is_moving_backward(csp_case_feed_kinematic_y.axis)
				)
			)
		THEN
			axis_stop(
		    	deceleration 	:= CONSTANTS.MAX_DECELERATION_MMpSEC2,
		    	jerk 			:= CONSTANTS.MAX_JERK_MMpSEC3,
		    	CONVERSION_this := csp_case_feed_kinematic_y.axis);
			fsm_next_status	:= CSP_CASE_FEED_KINEMATIC_STATUS_STOP_MCS2;
		END_IF
	
		
	CSP_CASE_FEED_KINEMATIC_STATUS_MOVE_MCS2:
	
		axis_move_absolute(
			position 		:= y_phase_position,
			velocity 		:= y_move_speed,
			direction		:= AXIS_CURRENT_DIRECTION,
			acceleration 	:= CONSTANTS.MAX_ACCELERATION_MMpSEC2,
			deceleration 	:= CONSTANTS.MAX_DECELERATION_MMpSEC2,
			jerk 			:= CONSTANTS.MAX_JERK_MMpSEC3, 
			buffer_mode 	:= AXIS_BUFFER_MODE_BUFFERED,
			CONVERSION_this := csp_case_feed_kinematic_y.axis);
				
		IF	axis_is_absolute_moving(csp_case_feed_kinematic_y.axis)
		THEN
			fsm_next_status	:= CSP_CASE_FEED_KINEMATIC_STATUS_STOP_MCS2;
		END_IF
	
		
	CSP_CASE_FEED_KINEMATIC_STATUS_STOP_MCS2:
	
		IF	axis_is_standstill(csp_case_feed_kinematic_y.axis)
		THEN			
			fsm_next_status	:= CSP_CASE_FEED_KINEMATIC_STATUS_ENABLED;
		END_IF
	
		
	CSP_CASE_FEED_KINEMATIC_STATUS_JOG_MCS3:
	
		IF	NOT tilt_jog_plus
			AND
			NOT tilt_jog_minus
			AND
			NOT command_button_is_pressed(hmi_tilt_jog_plus_cbtn)
			AND
			NOT command_button_is_pressed(hmi_tilt_jog_minus_cbtn)
			AND
			(
				NOT hmi_tilt_pendant_active
				OR
				(
					NOT csp_main_jogManager.pendant_positive_cmd
					AND
					axis_is_moving_forward(csp_case_feed_kinematic_tilt.axis)
				)
				OR
				(
					NOT csp_main_jogManager.pendant_negative_cmd
					AND
					axis_is_moving_backward(csp_case_feed_kinematic_tilt.axis)
				)
			)
		THEN
			axis_stop(
		    	deceleration 	:= CONSTANTS.MAX_DECELERATION_MMpSEC2,
		    	jerk 			:= CONSTANTS.MAX_JERK_MMpSEC3,
		    	CONVERSION_this := csp_case_feed_kinematic_tilt.axis);
			fsm_next_status	:= CSP_CASE_FEED_KINEMATIC_STATUS_STOP_MCS3;
		END_IF
	
		
	CSP_CASE_FEED_KINEMATIC_STATUS_MOVE_MCS3:
	
		axis_move_absolute(
			position 		:= tilt_phase_position,
			velocity 		:= tilt_move_speed,
			direction		:= AXIS_CURRENT_DIRECTION,
			acceleration 	:= CONSTANTS.MAX_ACCELERATION_MMpSEC2,
			deceleration 	:= CONSTANTS.MAX_DECELERATION_MMpSEC2,
			jerk 			:= CONSTANTS.MAX_JERK_MMpSEC3, 
			buffer_mode 	:= AXIS_BUFFER_MODE_BUFFERED,
			CONVERSION_this := csp_case_feed_kinematic_tilt.axis);
				
		IF	axis_is_absolute_moving(csp_case_feed_kinematic_tilt.axis)
		THEN
			fsm_next_status	:= CSP_CASE_FEED_KINEMATIC_STATUS_STOP_MCS3;
		END_IF
		
		
	CSP_CASE_FEED_KINEMATIC_STATUS_STOP_MCS3:
	
		IF	axis_is_standstill(csp_case_feed_kinematic_tilt.axis)
		THEN			
			fsm_next_status	:= CSP_CASE_FEED_KINEMATIC_STATUS_ENABLED;
		END_IF
		
		
	CSP_CASE_FEED_KINEMATIC_STATUS_PHASE_REQUEST:
	
		IF 	move_kinematic
		THEN
			x_phase_distance := ABS(axis_get_actual_incremental_position(csp_case_feed_kinematic_x.axis)-x_phase_position);
			y_phase_distance := ABS(axis_get_actual_incremental_position(csp_case_feed_kinematic_y.axis)-y_phase_position);
			phase_move_time := SQRT(x_phase_distance*x_phase_distance + y_phase_distance*y_phase_distance)/phase_move_speed;
			IF	phase_move_time > 0
			THEN 							
				x_phase_move_speed := SEL(x_phase_distance > 1, x_move_speed, x_phase_distance/phase_move_time);
				y_phase_move_speed := SEL(y_phase_distance > 1, y_move_speed, y_phase_distance/phase_move_time);
			ELSE
				x_phase_move_speed := x_move_speed;
				y_phase_move_speed := y_move_speed;
			END_IF
	
			axis_move_absolute(
				position 		:= x_phase_position,
				velocity 		:= x_phase_move_speed, //x_move_speed,
				direction		:= AXIS_CURRENT_DIRECTION,
				acceleration 	:= CONSTANTS.MAX_ACCELERATION_MMpSEC2,
				deceleration 	:= CONSTANTS.MAX_DECELERATION_MMpSEC2,
				jerk 			:= CONSTANTS.MAX_JERK_MMpSEC3, 
				buffer_mode 	:= AXIS_BUFFER_MODE_BUFFERED,
				CONVERSION_this := csp_case_feed_kinematic_x.axis); 
						
			axis_move_absolute(
				position 		:= y_phase_position,
				velocity 		:= y_phase_move_speed, //y_move_speed,
				direction		:= AXIS_CURRENT_DIRECTION,
				acceleration 	:= CONSTANTS.MAX_ACCELERATION_MMpSEC2,
				deceleration 	:= CONSTANTS.MAX_DECELERATION_MMpSEC2,
				jerk 			:= CONSTANTS.MAX_JERK_MMpSEC3, 
				buffer_mode 	:= AXIS_BUFFER_MODE_BUFFERED,
				CONVERSION_this := csp_case_feed_kinematic_y.axis); 
			
			axis_move_absolute(
				position 		:= tilt_phase_position,
				velocity 		:= tilt_move_speed,
				direction		:= AXIS_CURRENT_DIRECTION,
				acceleration 	:= CONSTANTS.MAX_ACCELERATION_MMpSEC2,
				deceleration 	:= CONSTANTS.MAX_DECELERATION_MMpSEC2,
				jerk 			:= CONSTANTS.MAX_JERK_MMpSEC3, 
				buffer_mode 	:= AXIS_BUFFER_MODE_BUFFERED,
				CONVERSION_this := csp_case_feed_kinematic_tilt.axis); 
			
			IF 	axis_is_absolute_moving(csp_case_feed_kinematic_x.axis)
				AND
				axis_is_absolute_moving(csp_case_feed_kinematic_y.axis)
				AND
				axis_is_absolute_moving(csp_case_feed_kinematic_tilt.axis)
			THEN
				fsm_next_status	:= CSP_CASE_FEED_KINEMATIC_STATUS_PHASING;
			END_IF
		ELSE
			axis_move_absolute(
				position 		:= elbow_phase_position,
				velocity 		:= elbow_move_speed,
				direction		:= AXIS_CURRENT_DIRECTION,
				acceleration 	:= CONSTANTS.MAX_ACCELERATION_MMpSEC2,
				deceleration 	:= CONSTANTS.MAX_DECELERATION_MMpSEC2,
				jerk 			:= CONSTANTS.MAX_JERK_MMpSEC3, 
				buffer_mode 	:= AXIS_BUFFER_MODE_BUFFERED,
				CONVERSION_this := csp_case_feed_arm_elbow.axis); 
			
			 axis_move_absolute(
				position 		:= shoulder_phase_position,
				velocity 		:= shoulder_move_speed,
				direction		:= AXIS_CURRENT_DIRECTION,
				acceleration 	:= CONSTANTS.MAX_ACCELERATION_MMpSEC2,
				deceleration 	:= CONSTANTS.MAX_DECELERATION_MMpSEC2,
				jerk 			:= CONSTANTS.MAX_JERK_MMpSEC3, 
				buffer_mode 	:= AXIS_BUFFER_MODE_BUFFERED,
				CONVERSION_this := csp_case_feed_arm_shoulder.axis); 
			
			axis_move_absolute(
				position 		:= wrist_phase_position,
				velocity 		:= wrist_move_speed,
				direction		:= AXIS_CURRENT_DIRECTION,
				acceleration 	:= CONSTANTS.MAX_ACCELERATION_MMpSEC2,
				deceleration 	:= CONSTANTS.MAX_DECELERATION_MMpSEC2,
				jerk 			:= CONSTANTS.MAX_JERK_MMpSEC3, 
				buffer_mode 	:= AXIS_BUFFER_MODE_BUFFERED,
				CONVERSION_this := csp_case_feed_arm_wrist.axis); 
			
			IF 	axis_is_absolute_moving(csp_case_feed_arm_elbow.axis)
				AND
				axis_is_absolute_moving(csp_case_feed_arm_shoulder.axis)
				AND
				axis_is_absolute_moving(csp_case_feed_arm_wrist.axis)
			THEN
				fsm_next_status	:= CSP_CASE_FEED_KINEMATIC_STATUS_PHASING;
			END_IF
		END_IF
		
		
	CSP_CASE_FEED_KINEMATIC_STATUS_PHASING:
	
		IF 	move_kinematic
		THEN
			IF 	axis_is_standstill(csp_case_feed_kinematic_x.axis)
				AND
				axis_is_standstill(csp_case_feed_kinematic_y.axis)
				AND
				axis_is_standstill(csp_case_feed_kinematic_tilt.axis)
			THEN
				IF	engage_enable
				THEN
					fsm_next_status	:= CSP_CASE_FEED_KINEMATIC_STATUS_READY_TO_ENGAGE;
				ELSE
					phase_request := FALSE;
					fsm_next_status	:= CSP_CASE_FEED_KINEMATIC_STATUS_ENABLED;
				END_IF
			END_IF
		ELSE
			IF 	axis_is_standstill(csp_case_feed_arm_elbow.axis)
				AND
				axis_is_standstill(csp_case_feed_arm_shoulder.axis)
				AND
				axis_is_standstill(csp_case_feed_arm_wrist.axis)
			THEN
				fsm_next_status	:= CSP_CASE_FEED_KINEMATIC_STATUS_PHASED;
			END_IF
		END_IF
		
		
	CSP_CASE_FEED_KINEMATIC_STATUS_PHASED:
	
		IF 	enable_kinematic
		THEN		
			kin_config_execute := TRUE;
			kin_config_cartesian_mode := TRUE;
			IF	fbConfigKinGroup.bDone
			THEN
				kin_config_execute := FALSE;	
				IF	move_kinematic
				THEN
					fsm_next_status	:= CSP_CASE_FEED_KINEMATIC_STATUS_PHASE_REQUEST;
				ELSE
					fsm_next_status	:= CSP_CASE_FEED_KINEMATIC_STATUS_READY_TO_ENGAGE;
				END_IF				
			END_IF
		END_IF
		
		
	CSP_CASE_FEED_KINEMATIC_STATUS_READY_TO_ENGAGE:
	
		move_kinematic := TRUE;		
		IF 	engage_enable 
			AND
			motorization_manager_is_starting(csp_main_motorization_manager.motm)					
		THEN			
			fsm_next_status := CSP_CASE_FEED_KINEMATIC_STATUS_CAM_ENGAGED_REQ;
		ELSIF NOT phase_request
		THEN
			fsm_next_status := CSP_CASE_FEED_KINEMATIC_STATUS_ENABLED;
		END_IF
				
		
	CSP_CASE_FEED_KINEMATIC_STATUS_CAM_ENGAGED_REQ:
	
		axis_engage_cam(
			cam_id 				:= CASE_FEED_KINEMATIC_X_RUN_CAM,
			master_engage_mode 	:= AXIS_CAM_ENGAGE_RELATIVE,
			slave_engage_mode 	:= AXIS_CAM_ENGAGE_RELATIVE,
			activation_mode 	:= AXIS_CAM_ACTIVATION_AT_MASTER_POSITION,
			activation_position	:= (axis_get_actual_modulo_turns(csp_case_virtualMaster.axis)+1.0)*axis_get_modulo(csp_case_virtualMaster.axis),
			master_scaling_mode	:= AXIS_CAM_SCALING_MODE_USER_DEFINED,
			slave_scaling_mode	:= AXIS_CAM_SCALING_MODE_AUTOOFFSET,
			master_offset 		:= 0,
			slave_offset 		:= 0,
			master_scaling 		:= master_scaling_deg,
			slave_scaling 		:= x_scaling_mm,
			interpolation_type 	:= AXIS_CAM_INTERPOLATION_SYSTEM_DEFAULT,
			master 				:= csp_case_virtualMaster.axis,
			CONVERSION_this 	:= csp_case_feed_kinematic_x.axis);
		x_old_scaling_mm := x_scaling_mm;
		
		axis_engage_cam(
			cam_id 				:= CASE_FEED_KINEMATIC_Y_RUN_CAM,
			master_engage_mode 	:= AXIS_CAM_ENGAGE_RELATIVE,
			slave_engage_mode 	:= AXIS_CAM_ENGAGE_RELATIVE,
			activation_mode 	:= AXIS_CAM_ACTIVATION_AT_MASTER_POSITION,
			activation_position	:= (axis_get_actual_modulo_turns(csp_case_virtualMaster.axis)+1.0)*axis_get_modulo(csp_case_virtualMaster.axis),
			master_scaling_mode	:= AXIS_CAM_SCALING_MODE_USER_DEFINED,
			slave_scaling_mode	:= AXIS_CAM_SCALING_MODE_AUTOOFFSET,
			master_offset 		:= 0,
			slave_offset 		:= 0,
			master_scaling 		:= master_scaling_deg,
			slave_scaling 		:= y_scaling_mm,
			interpolation_type 	:= AXIS_CAM_INTERPOLATION_SYSTEM_DEFAULT,
			master 				:= csp_case_virtualMaster.axis,
			CONVERSION_this 	:= csp_case_feed_kinematic_y.axis);
		y_old_scaling_mm := y_scaling_mm;
		
		axis_engage_cam(
			cam_id 				:= CASE_FEED_KINEMATIC_TILT_RUN_CAM,
			master_engage_mode 	:= AXIS_CAM_ENGAGE_RELATIVE,
			slave_engage_mode 	:= AXIS_CAM_ENGAGE_RELATIVE,
			activation_mode 	:= AXIS_CAM_ACTIVATION_AT_MASTER_POSITION,
			activation_position	:= (axis_get_actual_modulo_turns(csp_case_virtualMaster.axis)+1.0)*axis_get_modulo(csp_case_virtualMaster.axis),
			master_scaling_mode	:= AXIS_CAM_SCALING_MODE_USER_DEFINED,
			slave_scaling_mode	:= AXIS_CAM_SCALING_MODE_AUTOOFFSET,
			master_offset 		:= 0,
			slave_offset 		:= 0,
			master_scaling 		:= master_scaling_deg,
			slave_scaling 		:= tilt_scaling_deg,
			interpolation_type 	:= AXIS_CAM_INTERPOLATION_SYSTEM_DEFAULT,
			master 				:= csp_case_virtualMaster.axis,
			CONVERSION_this 	:= csp_case_feed_kinematic_tilt.axis);
		tilt_old_scaling_deg := tilt_scaling_deg;
	
		IF	axis_is_cam_engaged(csp_case_feed_kinematic_x.axis)
			AND
			axis_is_cam_engaged(csp_case_feed_kinematic_y.axis)
			AND
			axis_is_cam_engaged(csp_case_feed_kinematic_tilt.axis)
		THEN
	   		fsm_next_status := CSP_CASE_FEED_KINEMATIC_STATUS_CAM_ENGAGED;
		END_IF;
		IF	motorization_manager_is_stopped(csp_main_motorization_manager.motm) OR
			(
				NOT motorization_manager_is_stopping(csp_main_motorization_manager.motm)
				AND
				motorization_manager_is_idle(csp_main_motorization_manager.motm)
			)		
		THEN
			fsm_next_status := CSP_CASE_FEED_KINEMATIC_STATUS_STOP_REQUEST;
		END_IF
		
		
	CSP_CASE_FEED_KINEMATIC_STATUS_CAM_ENGAGED:
	
		IF 	(ABS(x_scaling_mm-x_old_scaling_mm) > 1)
			OR
			(ABS(y_scaling_mm-y_old_scaling_mm) > 1)
			OR
			(ABS(tilt_scaling_deg-tilt_old_scaling_deg) > 1)
		THEN									
			fsm_next_status := CSP_CASE_FEED_KINEMATIC_STATUS_CAM_ENGAGED_REQ;
		END_IF
		IF	motorization_manager_is_stopped(csp_main_motorization_manager.motm) OR
			(
				NOT motorization_manager_is_stopping(csp_main_motorization_manager.motm)
				AND
				motorization_manager_is_idle(csp_main_motorization_manager.motm)
			)
		THEN
			fsm_next_status := CSP_CASE_FEED_KINEMATIC_STATUS_STOP_REQUEST;
		END_IF
		
		
	CSP_CASE_FEED_KINEMATIC_STATUS_STOP_REQUEST:	
			
		axis_stop(
		    deceleration 	:= CONSTANTS.MAX_DECELERATION_MMpSEC2,
		    jerk 			:= CONSTANTS.MAX_JERK_MMpSEC3,
		    CONVERSION_this := csp_case_feed_kinematic_x.axis);
			
		axis_stop(
		    deceleration 	:= CONSTANTS.MAX_DECELERATION_MMpSEC2,
		    jerk 			:= CONSTANTS.MAX_JERK_MMpSEC3,
		    CONVERSION_this := csp_case_feed_kinematic_y.axis);
			
		axis_stop(
		    deceleration 	:= CONSTANTS.MAX_DECELERATION_MMpSEC2,
		    jerk 			:= CONSTANTS.MAX_JERK_MMpSEC3,
		    CONVERSION_this := csp_case_feed_kinematic_tilt.axis);

		IF 	(
				axis_is_standstill(csp_case_feed_kinematic_x.axis)
				OR
				NOT axis_is_ok(FALSE, csp_case_feed_kinematic_x.axis)
				OR
				axis_is_disabled(csp_case_feed_kinematic_x.axis)
			)
			AND
			(
				axis_is_standstill(csp_case_feed_kinematic_y.axis)
				OR
				NOT axis_is_ok(FALSE, csp_case_feed_kinematic_y.axis)
				OR
				axis_is_disabled(csp_case_feed_kinematic_y.axis)
			)
			AND
			(
				axis_is_standstill(csp_case_feed_kinematic_tilt.axis)
				OR
				NOT axis_is_ok(FALSE, csp_case_feed_kinematic_tilt.axis)
				OR
				axis_is_disabled(csp_case_feed_kinematic_tilt.axis)
			)
		THEN
			IF	fsm_enable_condition
			THEN
				fsm_next_status := CSP_CASE_FEED_KINEMATIC_STATUS_READY_TO_ENGAGE;
			ELSE
				fsm_next_status := CSP_CASE_FEED_KINEMATIC_STATUS_DISABLE_REQUEST;
			END_IF
		END_IF		

		
	CSP_CASE_FEED_KINEMATIC_STATUS_DISABLE_REQUEST:
	
		IF	disable_kinematic
		THEN
			kin_config_execute := TRUE;
			kin_config_cartesian_mode := FALSE;			
			fsm_next_status := CSP_CASE_FEED_KINEMATIC_STATUS_DISABLING_KINEMATIC;
		ELSE
			fsm_next_status := CSP_CASE_FEED_KINEMATIC_STATUS_DISABLING_AXIS;
		END_IF
		
		
	CSP_CASE_FEED_KINEMATIC_STATUS_DISABLING_KINEMATIC:
	
		IF	fbConfigKinGroup.bDone
			OR
			fbConfigKinGroup.bError			
        THEN
			kin_config_execute := FALSE;
			fsm_next_status := CSP_CASE_FEED_KINEMATIC_STATUS_DISABLING_AXIS;
		END_IF
		
		
	CSP_CASE_FEED_KINEMATIC_STATUS_DISABLING_AXIS:	
	
   		axis_disable(csp_case_feed_arm_elbow.axis);
		axis_disable(csp_case_feed_arm_shoulder.axis);
		axis_disable(csp_case_feed_arm_wrist.axis);
		axis_disable(csp_case_feed_kinematic_x.axis);
		axis_disable(csp_case_feed_kinematic_y.axis);
		axis_disable(csp_case_feed_kinematic_tilt.axis);
   		fsm_next_status := CSP_CASE_FEED_KINEMATIC_STATUS_DISABLING;

		
	CSP_CASE_FEED_KINEMATIC_STATUS_DISABLING:
	
        IF	axis_is_disabled(csp_case_feed_arm_elbow.axis)
			AND
			axis_is_disabled(csp_case_feed_arm_shoulder.axis)
			AND
			axis_is_disabled(csp_case_feed_arm_wrist.axis)
			AND
			axis_is_disabled(csp_case_feed_kinematic_x.axis)
			AND
			axis_is_disabled(csp_case_feed_kinematic_y.axis)
			AND			
			axis_is_disabled(csp_case_feed_kinematic_tilt.axis)			
        THEN			
            fsm_next_status := CSP_CASE_FEED_KINEMATIC_STATUS_DISABLED;
        END_IF
		
END_CASE

IF 	NOT debug_state_machine
	OR
	debug_state_machine_one_step
THEN
	fsm_status := fsm_next_status;
	debug_state_machine_one_step := FALSE;
END_IF

memo_cartesian_mode_request := ext_cartesian_mode_request;
memo_phase_request := ext_phase_request;
memo_stop_request := ext_stop_request;
(************************************************************************)

_handle_messages();

_write_output();

ACTION _handle_messages:
IF	fbConfigKinGroup.bError
THEN
	process_message_set(
		errorID_1			:= fbConfigKinGroup.nErrorId,
		errorID_2			:= 0,
		errorID_3			:= 0,
		CONVERSION_this 	:= kin_config_group_aem);
END_IF
END_ACTION

ACTION _handle_process_test:
;
END_ACTION

ACTION _hmi_management:
//Joint/Cartesian selection
command_button_led_set_status(
	status				:= SEL(fbConfigKinGroup.bBusy, HMI_OBJECT_STATUS_ON, HMI_OBJECT_STATUS_FAST_BLINKING), 		
	CONVERSION_this		:= hmi_joint_cartesian_mode_cbtn);
command_button_led_set_color(
	color				:= SEL(kin_config_cartesian_mode, HMI_LED_COLOR_YELLOW, HMI_LED_COLOR_GREEN), 		
	CONVERSION_this		:= hmi_joint_cartesian_mode_cbtn);

//Phase request
command_button_led_set_status(
	status				:= HMI_OBJECT_STATUS_ON, 		
	CONVERSION_this		:= hmi_phase_request_cbtn);
command_button_led_set_color(
	color				:= SEL(phase_request, HMI_LED_COLOR_YELLOW, HMI_LED_COLOR_GREEN), 		
	CONVERSION_this		:= hmi_phase_request_cbtn);
IF	command_button_is_pressed(hmi_phase_request_cbtn)
	AND
	NOT hmi_phase_request_cbtn_is_pressed
THEN
	phase_request		:= NOT phase_request;
END_IF	
hmi_phase_request_cbtn_is_pressed := command_button_is_pressed(hmi_phase_request_cbtn);

//Elbow command
command_button_led_set_status(
	status				:= HMI_OBJECT_STATUS_ON, 		
	CONVERSION_this		:= hmi_elbow_jog_plus_cbtn);
command_button_led_set_color(
	color				:= SEL(elbow_jog_plus, HMI_LED_COLOR_GREY, HMI_LED_COLOR_GREEN), 		
	CONVERSION_this		:= hmi_elbow_jog_plus_cbtn);
command_button_led_set_status(
	status				:= HMI_OBJECT_STATUS_ON, 		
	CONVERSION_this		:= hmi_elbow_jog_minus_cbtn);
command_button_led_set_color(
	color				:= SEL(elbow_jog_minus, HMI_LED_COLOR_GREY, HMI_LED_COLOR_GREEN), 		
	CONVERSION_this		:= hmi_elbow_jog_minus_cbtn);
command_button_led_set_status(
	status				:= HMI_OBJECT_STATUS_ON, 		
	CONVERSION_this		:= hmi_elbow_phase_move_cbtn);
command_button_led_set_color(
	color				:= SEL(axis_is_moving(csp_case_feed_arm_elbow.axis), HMI_LED_COLOR_GREY, HMI_LED_COLOR_GREEN), 		
	CONVERSION_this		:= hmi_elbow_phase_move_cbtn);
command_button_led_set_status(
	status				:= HMI_OBJECT_STATUS_ON, 		
	CONVERSION_this		:= hmi_elbow_activate_pendant_cbtn);
command_button_led_set_color(
	color				:= SEL(hmi_elbow_pendant_active, HMI_LED_COLOR_GREY, HMI_LED_COLOR_GREEN), 		
	CONVERSION_this		:= hmi_elbow_activate_pendant_cbtn);
IF	command_button_is_pressed(hmi_elbow_activate_pendant_cbtn)
	AND
	NOT hmi_elbow_activate_pendant_cbtn_is_pressed
THEN
	hmi_elbow_pendant_active := NOT hmi_elbow_pendant_active;
	IF	hmi_elbow_pendant_active
	THEN
		jog_manager_reset_pendant_active(csp_main_jogManager.jog_manager_real);
		hmi_shoulder_pendant_active := FALSE;
		hmi_wrist_pendant_active := FALSE;
		hmi_x_pendant_active := FALSE;
		hmi_y_pendant_active := FALSE;
		hmi_tilt_pendant_active := FALSE;
	END_IF
END_IF
hmi_elbow_activate_pendant_cbtn_is_pressed := command_button_is_pressed(hmi_elbow_activate_pendant_cbtn);

//Shoulder command
command_button_led_set_status(
	status				:= HMI_OBJECT_STATUS_ON, 		
	CONVERSION_this		:= hmi_shoulder_jog_plus_cbtn);
command_button_led_set_color(
	color				:= SEL(shoulder_jog_plus, HMI_LED_COLOR_GREY, HMI_LED_COLOR_GREEN), 		
	CONVERSION_this		:= hmi_shoulder_jog_plus_cbtn);
command_button_led_set_status(
	status				:= HMI_OBJECT_STATUS_ON, 		
	CONVERSION_this		:= hmi_shoulder_jog_minus_cbtn);
command_button_led_set_color(
	color				:= SEL(shoulder_jog_minus, HMI_LED_COLOR_GREY, HMI_LED_COLOR_GREEN), 		
	CONVERSION_this		:= hmi_shoulder_jog_minus_cbtn);
command_button_led_set_status(
	status				:= HMI_OBJECT_STATUS_ON, 		
	CONVERSION_this		:= hmi_shoulder_phase_move_cbtn);
command_button_led_set_color(
	color				:= SEL(axis_is_moving(csp_case_feed_arm_shoulder.axis), HMI_LED_COLOR_GREY, HMI_LED_COLOR_GREEN), 		
	CONVERSION_this		:= hmi_shoulder_phase_move_cbtn);
command_button_led_set_status(
	status				:= HMI_OBJECT_STATUS_ON, 		
	CONVERSION_this		:= hmi_shoulder_activate_pendant_cbtn);
command_button_led_set_color(
	color				:= SEL(hmi_shoulder_pendant_active, HMI_LED_COLOR_GREY, HMI_LED_COLOR_GREEN), 		
	CONVERSION_this		:= hmi_shoulder_activate_pendant_cbtn);
IF	command_button_is_pressed(hmi_shoulder_activate_pendant_cbtn)
	AND
	NOT hmi_shoulder_activate_pendant_cbtn_is_pressed
THEN
	hmi_shoulder_pendant_active := NOT hmi_shoulder_pendant_active;
	IF	hmi_shoulder_pendant_active
	THEN
		jog_manager_reset_pendant_active(csp_main_jogManager.jog_manager_real);
		hmi_elbow_pendant_active := FALSE;
		hmi_wrist_pendant_active := FALSE;
		hmi_x_pendant_active := FALSE;
		hmi_y_pendant_active := FALSE;
		hmi_tilt_pendant_active := FALSE;
	END_IF
END_IF
hmi_shoulder_activate_pendant_cbtn_is_pressed := command_button_is_pressed(hmi_shoulder_activate_pendant_cbtn);

//Wrist command
command_button_led_set_status(
	status				:= HMI_OBJECT_STATUS_ON, 		
	CONVERSION_this		:= hmi_wrist_jog_plus_cbtn);
command_button_led_set_color(
	color				:= SEL(wrist_jog_plus, HMI_LED_COLOR_GREY, HMI_LED_COLOR_GREEN), 		
	CONVERSION_this		:= hmi_wrist_jog_plus_cbtn);
command_button_led_set_status(
	status				:= HMI_OBJECT_STATUS_ON, 		
	CONVERSION_this		:= hmi_wrist_jog_minus_cbtn);
command_button_led_set_color(
	color				:= SEL(wrist_jog_minus, HMI_LED_COLOR_GREY, HMI_LED_COLOR_GREEN), 		
	CONVERSION_this		:= hmi_wrist_jog_minus_cbtn);
command_button_led_set_status(
	status				:= HMI_OBJECT_STATUS_ON, 		
	CONVERSION_this		:= hmi_wrist_phase_move_cbtn);
command_button_led_set_color(
	color				:= SEL(axis_is_moving(csp_case_feed_arm_wrist.axis), HMI_LED_COLOR_GREY, HMI_LED_COLOR_GREEN), 		
	CONVERSION_this		:= hmi_wrist_phase_move_cbtn);
command_button_led_set_status(
	status				:= HMI_OBJECT_STATUS_ON, 		
	CONVERSION_this		:= hmi_wrist_activate_pendant_cbtn);
command_button_led_set_color(
	color				:= SEL(hmi_wrist_pendant_active, HMI_LED_COLOR_GREY, HMI_LED_COLOR_GREEN), 		
	CONVERSION_this		:= hmi_wrist_activate_pendant_cbtn);
IF	command_button_is_pressed(hmi_wrist_activate_pendant_cbtn)
	AND
	NOT hmi_wrist_activate_pendant_cbtn_is_pressed
THEN
	hmi_wrist_pendant_active := NOT hmi_wrist_pendant_active;
	IF	hmi_wrist_pendant_active
	THEN
		jog_manager_reset_pendant_active(csp_main_jogManager.jog_manager_real);
		hmi_shoulder_pendant_active := FALSE;
		hmi_elbow_pendant_active := FALSE;
		hmi_x_pendant_active := FALSE;
		hmi_y_pendant_active := FALSE;
		hmi_tilt_pendant_active := FALSE;
	END_IF
END_IF
hmi_wrist_activate_pendant_cbtn_is_pressed := command_button_is_pressed(hmi_wrist_activate_pendant_cbtn);

//X command
command_button_led_set_status(
	status				:= HMI_OBJECT_STATUS_ON, 		
	CONVERSION_this		:= hmi_x_jog_plus_cbtn);
command_button_led_set_color(
	color				:= SEL(x_jog_plus, HMI_LED_COLOR_GREY, HMI_LED_COLOR_GREEN), 		
	CONVERSION_this		:= hmi_x_jog_plus_cbtn);
command_button_led_set_status(
	status				:= HMI_OBJECT_STATUS_ON, 		
	CONVERSION_this		:= hmi_x_jog_minus_cbtn);
command_button_led_set_color(
	color				:= SEL(x_jog_minus, HMI_LED_COLOR_GREY, HMI_LED_COLOR_GREEN), 		
	CONVERSION_this		:= hmi_x_jog_minus_cbtn);
command_button_led_set_status(
	status				:= HMI_OBJECT_STATUS_ON, 		
	CONVERSION_this		:= hmi_x_phase_move_cbtn);
command_button_led_set_color(
	color				:= SEL(axis_is_moving(csp_case_feed_kinematic_x.axis), HMI_LED_COLOR_GREY, HMI_LED_COLOR_GREEN), 		
	CONVERSION_this		:= hmi_x_phase_move_cbtn);
command_button_led_set_status(
	status				:= HMI_OBJECT_STATUS_ON, 		
	CONVERSION_this		:= hmi_x_activate_pendant_cbtn);
command_button_led_set_color(
	color				:= SEL(hmi_x_pendant_active, HMI_LED_COLOR_GREY, HMI_LED_COLOR_GREEN), 		
	CONVERSION_this		:= hmi_x_activate_pendant_cbtn);
IF	command_button_is_pressed(hmi_x_activate_pendant_cbtn)
	AND
	NOT hmi_x_activate_pendant_cbtn_is_pressed
THEN
	hmi_x_pendant_active := NOT hmi_x_pendant_active;
	IF	hmi_x_pendant_active
	THEN
		jog_manager_reset_pendant_active(csp_main_jogManager.jog_manager_real);
		hmi_shoulder_pendant_active := FALSE;
		hmi_elbow_pendant_active := FALSE;
		hmi_wrist_pendant_active := FALSE;
		hmi_y_pendant_active := FALSE;
		hmi_tilt_pendant_active := FALSE;
	END_IF
END_IF
hmi_x_activate_pendant_cbtn_is_pressed := command_button_is_pressed(hmi_x_activate_pendant_cbtn);

//Y command
command_button_led_set_status(
	status				:= HMI_OBJECT_STATUS_ON, 		
	CONVERSION_this		:= hmi_y_jog_plus_cbtn);
command_button_led_set_color(
	color				:= SEL(y_jog_plus, HMI_LED_COLOR_GREY, HMI_LED_COLOR_GREEN), 		
	CONVERSION_this		:= hmi_y_jog_plus_cbtn);
command_button_led_set_status(
	status				:= HMI_OBJECT_STATUS_ON, 		
	CONVERSION_this		:= hmi_y_jog_minus_cbtn);
command_button_led_set_color(
	color				:= SEL(y_jog_minus, HMI_LED_COLOR_GREY, HMI_LED_COLOR_GREEN), 		
	CONVERSION_this		:= hmi_y_jog_minus_cbtn);
command_button_led_set_status(
	status				:= HMI_OBJECT_STATUS_ON, 		
	CONVERSION_this		:= hmi_y_phase_move_cbtn);
command_button_led_set_color(
	color				:= SEL(axis_is_moving(csp_case_feed_kinematic_y.axis), HMI_LED_COLOR_GREY, HMI_LED_COLOR_GREEN), 		
	CONVERSION_this		:= hmi_y_phase_move_cbtn);
command_button_led_set_status(
	status				:= HMI_OBJECT_STATUS_ON, 		
	CONVERSION_this		:= hmi_y_activate_pendant_cbtn);
command_button_led_set_color(
	color				:= SEL(hmi_y_pendant_active, HMI_LED_COLOR_GREY, HMI_LED_COLOR_GREEN), 		
	CONVERSION_this		:= hmi_y_activate_pendant_cbtn);
IF	command_button_is_pressed(hmi_y_activate_pendant_cbtn)
	AND
	NOT hmi_y_activate_pendant_cbtn_is_pressed
THEN
	hmi_y_pendant_active := NOT hmi_y_pendant_active;
	IF	hmi_y_pendant_active
	THEN
		jog_manager_reset_pendant_active(csp_main_jogManager.jog_manager_real);
		hmi_shoulder_pendant_active := FALSE;
		hmi_elbow_pendant_active := FALSE;
		hmi_wrist_pendant_active := FALSE;
		hmi_x_pendant_active := FALSE;
		hmi_tilt_pendant_active := FALSE;
	END_IF
END_IF
hmi_y_activate_pendant_cbtn_is_pressed := command_button_is_pressed(hmi_y_activate_pendant_cbtn);

//Tilt command
command_button_led_set_status(
	status				:= HMI_OBJECT_STATUS_ON, 		
	CONVERSION_this		:= hmi_tilt_jog_plus_cbtn);
command_button_led_set_color(
	color				:= SEL(tilt_jog_plus, HMI_LED_COLOR_GREY, HMI_LED_COLOR_GREEN), 		
	CONVERSION_this		:= hmi_tilt_jog_plus_cbtn);
command_button_led_set_status(
	status				:= HMI_OBJECT_STATUS_ON, 		
	CONVERSION_this		:= hmi_tilt_jog_minus_cbtn);
command_button_led_set_color(
	color				:= SEL(tilt_jog_minus, HMI_LED_COLOR_GREY, HMI_LED_COLOR_GREEN), 		
	CONVERSION_this		:= hmi_tilt_jog_minus_cbtn);
command_button_led_set_status(
	status				:= HMI_OBJECT_STATUS_ON, 		
	CONVERSION_this		:= hmi_tilt_phase_move_cbtn);
command_button_led_set_color(
	color				:= SEL(axis_is_moving(csp_case_feed_kinematic_tilt.axis), HMI_LED_COLOR_GREY, HMI_LED_COLOR_GREEN), 		
	CONVERSION_this		:= hmi_tilt_phase_move_cbtn);
command_button_led_set_status(
	status				:= HMI_OBJECT_STATUS_ON, 		
	CONVERSION_this		:= hmi_tilt_activate_pendant_cbtn);
command_button_led_set_color(
	color				:= SEL(hmi_tilt_pendant_active, HMI_LED_COLOR_GREY, HMI_LED_COLOR_GREEN), 		
	CONVERSION_this		:= hmi_tilt_activate_pendant_cbtn);
IF	command_button_is_pressed(hmi_tilt_activate_pendant_cbtn)
	AND
	NOT hmi_tilt_activate_pendant_cbtn_is_pressed
THEN
	hmi_tilt_pendant_active := NOT hmi_tilt_pendant_active;
	IF	hmi_tilt_pendant_active
	THEN
		jog_manager_reset_pendant_active(csp_main_jogManager.jog_manager_real);
		hmi_shoulder_pendant_active := FALSE;
		hmi_elbow_pendant_active := FALSE;
		hmi_wrist_pendant_active := FALSE;
		hmi_x_pendant_active := FALSE;
		hmi_y_pendant_active := FALSE;
	END_IF
END_IF
hmi_tilt_activate_pendant_cbtn_is_pressed := command_button_is_pressed(hmi_tilt_activate_pendant_cbtn);

//External pendant selection
hmi_pendant_active := 
	hmi_elbow_pendant_active
	OR
	hmi_shoulder_pendant_active
	OR
	hmi_wrist_pendant_active
	OR
	hmi_x_pendant_active
	OR
	hmi_y_pendant_active
	OR
	hmi_tilt_pendant_active;
IF	hmi_pendant_active
	AND
	jog_manager_is_pendant_active(csp_main_jogManager.jog_manager_real)
THEN
	hmi_elbow_pendant_active := FALSE;
	hmi_shoulder_pendant_active := FALSE;
	hmi_wrist_pendant_active := FALSE;
	hmi_x_pendant_active := FALSE;
	hmi_y_pendant_active := FALSE;
	hmi_tilt_pendant_active := FALSE;
END_IF

//Object status
hmi_graphic_object_set_status(
	status  			:= SEL(visu_disable_general_command, HMI_OBJECT_STATUS_ON, HMI_OBJECT_STATUS_LOCKED),
	CONVERSION_this    	:= hmi_enable_general_command_hgos);

hmi_graphic_object_set_status(
	status  			:= SEL(kin_config_cartesian_mode, HMI_OBJECT_STATUS_ON, HMI_OBJECT_STATUS_INVISIBLE),
	CONVERSION_this    	:= hmi_enable_joint_hgos);

hmi_graphic_object_set_status(
	status  			:= SEL(NOT kin_config_cartesian_mode, HMI_OBJECT_STATUS_ON, HMI_OBJECT_STATUS_INVISIBLE),
	CONVERSION_this    	:= hmi_enable_cartesian_hgos);
	
hmi_graphic_object_set_status(
	status  			:= SEL(visu_disable_ACS_command, HMI_OBJECT_STATUS_ON, HMI_OBJECT_STATUS_LOCKED),
	CONVERSION_this    	:= hmi_enable_ACS_command_hgos);
	
hmi_graphic_object_set_status(
	status  			:= SEL(visu_disable_MCS_command, HMI_OBJECT_STATUS_ON, HMI_OBJECT_STATUS_LOCKED),
	CONVERSION_this    	:= hmi_enable_MCS_command_hgos);
command_button_set_status(
	status				:= SEL(visu_disable_MCS_jog_mode OR hmi_x_pendant_active, HMI_OBJECT_STATUS_ON, HMI_OBJECT_STATUS_LOCKED),	
	CONVERSION_this    	:= hmi_x_jog_plus_cbtn);
command_button_set_status(
	status				:= SEL(visu_disable_MCS_jog_mode OR hmi_x_pendant_active, HMI_OBJECT_STATUS_ON, HMI_OBJECT_STATUS_LOCKED),	
	CONVERSION_this    	:= hmi_x_jog_minus_cbtn);
command_button_set_status(
	status				:= SEL(visu_disable_MCS_jog_mode OR hmi_y_pendant_active, HMI_OBJECT_STATUS_ON, HMI_OBJECT_STATUS_LOCKED),	
	CONVERSION_this    	:= hmi_y_jog_plus_cbtn);
command_button_set_status(
	status				:= SEL(visu_disable_MCS_jog_mode OR hmi_y_pendant_active, HMI_OBJECT_STATUS_ON, HMI_OBJECT_STATUS_LOCKED),	
	CONVERSION_this    	:= hmi_y_jog_minus_cbtn);
command_button_set_status(
	status				:= SEL(visu_disable_MCS_jog_mode OR hmi_tilt_pendant_active, HMI_OBJECT_STATUS_ON, HMI_OBJECT_STATUS_LOCKED),	
	CONVERSION_this    	:= hmi_tilt_jog_plus_cbtn);
command_button_set_status(
	status				:= SEL(visu_disable_MCS_jog_mode OR hmi_tilt_pendant_active, HMI_OBJECT_STATUS_ON, HMI_OBJECT_STATUS_LOCKED),	
	CONVERSION_this    	:= hmi_tilt_jog_minus_cbtn);
	
hmi_graphic_object_set_status(
	status  			:= SEL(visu_disable_ACS_jog_mode, HMI_OBJECT_STATUS_ON, HMI_OBJECT_STATUS_LOCKED),
	CONVERSION_this    	:= hmi_enable_ACS_jog_mode_hgos);
command_button_set_status(
	status				:= SEL(visu_disable_ACS_jog_mode OR hmi_elbow_pendant_active, HMI_OBJECT_STATUS_ON, HMI_OBJECT_STATUS_LOCKED),	
	CONVERSION_this    	:= hmi_elbow_jog_plus_cbtn);
command_button_set_status(
	status				:= SEL(visu_disable_ACS_jog_mode OR hmi_elbow_pendant_active, HMI_OBJECT_STATUS_ON, HMI_OBJECT_STATUS_LOCKED),	
	CONVERSION_this    	:= hmi_elbow_jog_minus_cbtn);
command_button_set_status(
	status				:= SEL(visu_disable_ACS_jog_mode OR hmi_shoulder_pendant_active, HMI_OBJECT_STATUS_ON, HMI_OBJECT_STATUS_LOCKED),	
	CONVERSION_this    	:= hmi_shoulder_jog_plus_cbtn);
command_button_set_status(
	status				:= SEL(visu_disable_ACS_jog_mode OR hmi_shoulder_pendant_active, HMI_OBJECT_STATUS_ON, HMI_OBJECT_STATUS_LOCKED),	
	CONVERSION_this    	:= hmi_shoulder_jog_minus_cbtn);
command_button_set_status(
	status				:= SEL(visu_disable_ACS_jog_mode OR hmi_wrist_pendant_active, HMI_OBJECT_STATUS_ON, HMI_OBJECT_STATUS_LOCKED),	
	CONVERSION_this    	:= hmi_wrist_jog_plus_cbtn);
command_button_set_status(
	status				:= SEL(visu_disable_ACS_jog_mode OR hmi_wrist_pendant_active, HMI_OBJECT_STATUS_ON, HMI_OBJECT_STATUS_LOCKED),	
	CONVERSION_this    	:= hmi_wrist_jog_minus_cbtn);
	
hmi_graphic_object_set_status(
	status  			:= SEL(visu_disable_MCS_jog_mode, HMI_OBJECT_STATUS_ON, HMI_OBJECT_STATUS_LOCKED),
	CONVERSION_this    	:= hmi_enable_MCS_jog_mode_hgos);
	
hmi_graphic_object_set_status(
	status  			:= SEL(visu_disable_phase_request, HMI_OBJECT_STATUS_ON, HMI_OBJECT_STATUS_LOCKED),
	CONVERSION_this    	:= hmi_enable_phase_request_hgos);
END_ACTION

ACTION _mode_manager:
IF process_mode_req_is_pending(prc)
THEN
    process_apply_mode_req_first_step(prc);
    CASE process_get_mode(prc) OF
        MODE_TO_ABSENT:
			;
        MODE_TO_INACTIVE:
			;
        MODE_TO_TEST:
			;
        MODE_TO_OPERATIONAL:
			;
    END_CASE
    process_apply_mode_req_second_step(prc);
END_IF
END_ACTION

ACTION _object_manager:
IF objects_initialization()
THEN
	sub_process_init(
		object_name					:= 'csp_case_feed_kinematic.prc', 
		process						:= csp_case_feed.prc, 
		CONVERSION_this				:= prc);
		
	prc_path 						:= process_get_path(prc);
		
	process_message_init(
		object_name					:= CONCAT(prc_path, '_kin_config_group_aem'), 
		behaviour					:= MESSAGE_BEHAVIOUR_EVENT,
		reset_timeout				:= 0,
		disableable					:= TRUE,
		individual_reset			:= FALSE,
		machine_reaction			:= MACHINE_REACTION_NORMAL_STOP,
		typology					:= MESSAGE_TYPOLOGY_ABNORMAL,
		process						:= prc,
		CONVERSION_this				:= kin_config_group_aem);
		
	//Parameter overwrite
	parameter_overwrite_lreal_init(
		object_name 				:= CONCAT(prc_path, '_elbow_phase_position_pow'),
		out_of_range				:= PARAMETER_OVERWRITE_OUT_OF_RANGE_NONE,
		parameter					:= elbow_phase_position,
		process						:= prc,
		CONVERSION_this 			:= elbow_phase_position_pow);
	
	parameter_overwrite_lreal_init(
		object_name 				:= CONCAT(prc_path, '_shoulder_phase_position_pow'),
		out_of_range				:= PARAMETER_OVERWRITE_OUT_OF_RANGE_NONE,
		parameter					:= shoulder_phase_position,
		process						:= prc,
		CONVERSION_this 			:= shoulder_phase_position_pow);
	
	parameter_overwrite_lreal_init(
		object_name 				:= CONCAT(prc_path, '_wrist_phase_position_pow'),
		out_of_range				:= PARAMETER_OVERWRITE_OUT_OF_RANGE_NONE,
		parameter					:= wrist_phase_position,
		process						:= prc,
		CONVERSION_this 			:= wrist_phase_position_pow);
		
	parameter_overwrite_lreal_init(
		object_name 				:= CONCAT(prc_path, '_x_phase_position_pow'),
		out_of_range				:= PARAMETER_OVERWRITE_OUT_OF_RANGE_NONE,
		parameter					:= x_phase_position,
		process						:= prc,
		CONVERSION_this 			:= x_phase_position_pow);
	
	parameter_overwrite_lreal_init(
		object_name 				:= CONCAT(prc_path, '_y_phase_position_pow'),
		out_of_range				:= PARAMETER_OVERWRITE_OUT_OF_RANGE_NONE,
		parameter					:= y_phase_position,
		process						:= prc,
		CONVERSION_this 			:= y_phase_position_pow);
	
	parameter_overwrite_lreal_init(
		object_name 				:= CONCAT(prc_path, '_tilt_phase_position_pow'),
		out_of_range				:= PARAMETER_OVERWRITE_OUT_OF_RANGE_NONE,
		parameter					:= tilt_phase_position,
		process						:= prc,
		CONVERSION_this 			:= tilt_phase_position_pow);
	
	//HMI custom page variable management	
	command_button_init(
	    object_name 				:= CONCAT(prc_path, '_hmi_joint_cartesian_mode_cbtn'),
	    process 					:= prc,
	    CONVERSION_this 			:= hmi_joint_cartesian_mode_cbtn);
	
	command_button_init(
	    object_name 				:= CONCAT(prc_path, '_hmi_phase_request_cbtn'),
	    process 					:= prc,
	    CONVERSION_this 			:= hmi_phase_request_cbtn);

		
	command_button_init(
	    object_name 				:= CONCAT(prc_path, '_hmi_elbow_jog_plus_cbtn'),
	    process 					:= prc,
	    CONVERSION_this 			:= hmi_elbow_jog_plus_cbtn);
	
	command_button_init(
	    object_name 				:= CONCAT(prc_path, '_hmi_elbow_jog_minus_cbtn'),
	    process 					:= prc,
	    CONVERSION_this 			:= hmi_elbow_jog_minus_cbtn);
	
	command_button_init(
	    object_name 				:= CONCAT(prc_path, '_hmi_elbow_phase_move_cbtn'),
	    process 					:= prc,
	    CONVERSION_this 			:= hmi_elbow_phase_move_cbtn);
	
	command_button_init(
	    object_name 				:= CONCAT(prc_path, '_hmi_elbow_copy_phase_cbtn'),
	    process 					:= prc,
	    CONVERSION_this 			:= hmi_elbow_copy_phase_cbtn);
		
	command_button_init(
	    object_name 				:= CONCAT(prc_path, '_hmi_elbow_activate_pendant_cbtn'),
	    process 					:= prc,
	    CONVERSION_this 			:= hmi_elbow_activate_pendant_cbtn);
	
				
	command_button_init(
	    object_name 				:= CONCAT(prc_path, '_hmi_shoulder_jog_plus_cbtn'),
	    process 					:= prc,
	    CONVERSION_this 			:= hmi_shoulder_jog_plus_cbtn);
	
	command_button_init(
	    object_name 				:= CONCAT(prc_path, '_hmi_shoulder_jog_minus_cbtn'),
	    process 					:= prc,
	    CONVERSION_this 			:= hmi_shoulder_jog_minus_cbtn);
	
	command_button_init(
	    object_name 				:= CONCAT(prc_path, '_hmi_shoulder_phase_move_cbtn'),
	    process 					:= prc,
	    CONVERSION_this 			:= hmi_shoulder_phase_move_cbtn);
	
	command_button_init(
	    object_name 				:= CONCAT(prc_path, '_hmi_shoulder_copy_phase_cbtn'),
	    process 					:= prc,
	    CONVERSION_this 			:= hmi_shoulder_copy_phase_cbtn);

	command_button_init(
	    object_name 				:= CONCAT(prc_path, '_hmi_shoulder_activate_pendant_cbtn'),
	    process 					:= prc,
	    CONVERSION_this 			:= hmi_shoulder_activate_pendant_cbtn);
	
	
	command_button_init(
	    object_name 				:= CONCAT(prc_path, '_hmi_wrist_jog_plus_cbtn'),
	    process 					:= prc,
	    CONVERSION_this 			:= hmi_wrist_jog_plus_cbtn);
	
	command_button_init(
	    object_name 				:= CONCAT(prc_path, '_hmi_wrist_jog_minus_cbtn'),
	    process 					:= prc,
	    CONVERSION_this 			:= hmi_wrist_jog_minus_cbtn);
	
	command_button_init(
	    object_name 				:= CONCAT(prc_path, '_hmi_wrist_phase_move_cbtn'),
	    process 					:= prc,
	    CONVERSION_this 			:= hmi_wrist_phase_move_cbtn);
	
	command_button_init(
	    object_name 				:= CONCAT(prc_path, '_hmi_wrist_copy_phase_cbtn'),
	    process 					:= prc,
	    CONVERSION_this 			:= hmi_wrist_copy_phase_cbtn);
	
	command_button_init(
	    object_name 				:= CONCAT(prc_path, '_hmi_wrist_activate_pendant_cbtn'),
	    process 					:= prc,
	    CONVERSION_this 			:= hmi_wrist_activate_pendant_cbtn);
	
		
	command_button_init(
	    object_name 				:= CONCAT(prc_path, '_hmi_x_jog_plus_cbtn'),
	    process 					:= prc,
	    CONVERSION_this 			:= hmi_x_jog_plus_cbtn);
	
	command_button_init(
	    object_name 				:= CONCAT(prc_path, '_hmi_x_jog_minus_cbtn'),
	    process 					:= prc,
	    CONVERSION_this 			:= hmi_x_jog_minus_cbtn);
	
	command_button_init(
	    object_name 				:= CONCAT(prc_path, '_hmi_x_phase_move_cbtn'),
	    process 					:= prc,
	    CONVERSION_this 			:= hmi_x_phase_move_cbtn);
	
	command_button_init(
	    object_name 				:= CONCAT(prc_path, '_hmi_x_copy_phase_cbtn'),
	    process 					:= prc,
	    CONVERSION_this 			:= hmi_x_copy_phase_cbtn);
	
	command_button_init(
	    object_name 				:= CONCAT(prc_path, '_hmi_x_activate_pendant_cbtn'),
	    process 					:= prc,
	    CONVERSION_this 			:= hmi_x_activate_pendant_cbtn);
	
		
	command_button_init(
	    object_name 				:= CONCAT(prc_path, '_hmi_y_jog_plus_cbtn'),
	    process 					:= prc,
	    CONVERSION_this 			:= hmi_y_jog_plus_cbtn);
	
	command_button_init(
	    object_name 				:= CONCAT(prc_path, '_hmi_y_jog_minus_cbtn'),
	    process 					:= prc,
	    CONVERSION_this 			:= hmi_y_jog_minus_cbtn);
	
	command_button_init(
	    object_name 				:= CONCAT(prc_path, '_hmi_y_phase_move_cbtn'),
	    process 					:= prc,
	    CONVERSION_this 			:= hmi_y_phase_move_cbtn);
	
	command_button_init(
	    object_name 				:= CONCAT(prc_path, '_hmi__copy_phase_cbtn'),
	    process 					:= prc,
	    CONVERSION_this 			:= hmi_y_copy_phase_cbtn);	
	
	command_button_init(
	    object_name 				:= CONCAT(prc_path, '_hmi_y_activate_pendant_cbtn'),
	    process 					:= prc,
	    CONVERSION_this 			:= hmi_y_activate_pendant_cbtn);
	
		
	command_button_init(
	    object_name 				:= CONCAT(prc_path, '_hmi_tilt_jog_plus_cbtn'),
	    process 					:= prc,
	    CONVERSION_this 			:= hmi_tilt_jog_plus_cbtn);
	
	command_button_init(
	    object_name 				:= CONCAT(prc_path, '_hmi_tilt_jog_minus_cbtn'),
	    process 					:= prc,
	    CONVERSION_this 			:= hmi_tilt_jog_minus_cbtn);
	
	command_button_init(
	    object_name 				:= CONCAT(prc_path, '_hmi_tilt_phase_move_cbtn'),
	    process 					:= prc,
	    CONVERSION_this 			:= hmi_tilt_phase_move_cbtn);
	
	command_button_init(
	    object_name 				:= CONCAT(prc_path, '_hmi_tilt_copy_phase_cbtn'),
	    process 					:= prc,
	    CONVERSION_this 			:= hmi_tilt_copy_phase_cbtn);	
	
	command_button_init(
	    object_name 				:= CONCAT(prc_path, '_hmi_tilt_activate_pendant_cbtn'),
	    process 					:= prc,
	    CONVERSION_this 			:= hmi_tilt_activate_pendant_cbtn);
	
		
	hmi_graphic_object_status_init(
        object_name         		:= CONCAT(prc_path, '_hmi_enable_general_command_hgos'),
        process             		:= prc,
        CONVERSION_this             := hmi_enable_general_command_hgos);
	
	hmi_graphic_object_status_init(
        object_name         		:= CONCAT(prc_path, '_hmi_enable_joint_hgos'),
        process             		:= prc,
        CONVERSION_this             := hmi_enable_joint_hgos);
	
	hmi_graphic_object_status_init(
        object_name         		:= CONCAT(prc_path, '_hmi_enable_cartesian_hgos'),
        process             		:= prc,
        CONVERSION_this             := hmi_enable_cartesian_hgos);
	
	hmi_graphic_object_status_init(
        object_name         		:= CONCAT(prc_path, '_hmi_enable_ACS_command_hgos'),
        process             		:= prc,
        CONVERSION_this             := hmi_enable_ACS_command_hgos);
	
	hmi_graphic_object_status_init(
        object_name         		:= CONCAT(prc_path, '_hmi_enable_MCS_command_hgos'),
        process             		:= prc,
        CONVERSION_this             := hmi_enable_MCS_command_hgos);
	
	hmi_graphic_object_status_init(
        object_name         		:= CONCAT(prc_path, '_hmi_enable_ACS_jog_mode_hgos'),
        process             		:= prc,
        CONVERSION_this             := hmi_enable_ACS_jog_mode_hgos);
	
	hmi_graphic_object_status_init(
        object_name         		:= CONCAT(prc_path, '_hmi_enable_MCS_jog_mode_hgos'),
        process             		:= prc,
        CONVERSION_this             := hmi_enable_MCS_jog_mode_hgos);
		
	hmi_graphic_object_status_init(
        object_name         		:= CONCAT(prc_path, '_hmi_enable_phase_request_hgos'),
        process             		:= prc,
        CONVERSION_this             := hmi_enable_phase_request_hgos);
	
		
	motorization_conditioner_init(
		object_name					:=	CONCAT(prc_path, '_kinematic_jog_on_motcond'),
		velocity_limit				:=	0.0,
		velocity_limit_active		:=	FALSE,
		idle_handshake_active		:=	FALSE,
		execute_handshake_active	:=	TRUE,
		hold_handshake_active		:=	FALSE,
		suspend_handshake_active	:=	FALSE,
		complete_handshake_active	:=	FALSE,
		abort_handshake_active		:=	FALSE,
		stop_handshake_active		:=	FALSE,
		origin						:=	MOTORIZATION_CONDITIONER_ORIGIN_INTERNAL,
		manager						:=	csp_main_motorization_manager.motm,
		process						:=	prc,
		CONVERSION_this				:=	kinematic_jog_on_motcond);
		
		
	process_message_init(
        object_name:= CONCAT(prc_path, '_Kinematic_tilt_error_aem'),
        behaviour:= MESSAGE_BEHAVIOUR_STATE,
        reset_timeout:= 0,
        disableable:= FALSE,
        individual_reset:= FALSE,
        machine_reaction:= MACHINE_REACTION_STOP_IN_PHASE_ONE, //MACHINE_REACTION_STOP_IN_PHASE_ONE,
        typology:=  MESSAGE_TYPOLOGY_ABNORMAL, //MESSAGE_TYPOLOGY_ABNORMAL,
        process:= prc,
        CONVERSION_this:= Kinematic_tilt_error_aem);	
END_IF

IF objects_running()
THEN
	process_cycle(prc);
	(*axis_cycle(axis);*)
	
	motorization_conditioner_cycle(kinematic_jog_on_motcond);
	
	command_button_cycle(hmi_joint_cartesian_mode_cbtn);
	command_button_cycle(hmi_phase_request_cbtn);
	command_button_cycle(hmi_elbow_jog_plus_cbtn);
	command_button_cycle(hmi_elbow_jog_minus_cbtn);
	command_button_cycle(hmi_elbow_phase_move_cbtn);
	command_button_cycle(hmi_elbow_copy_phase_cbtn);
	command_button_cycle(hmi_elbow_activate_pendant_cbtn);
	command_button_cycle(hmi_shoulder_jog_plus_cbtn);
	command_button_cycle(hmi_shoulder_jog_minus_cbtn);
	command_button_cycle(hmi_shoulder_phase_move_cbtn);
	command_button_cycle(hmi_shoulder_copy_phase_cbtn);
	command_button_cycle(hmi_shoulder_activate_pendant_cbtn);
	command_button_cycle(hmi_wrist_jog_plus_cbtn);
	command_button_cycle(hmi_wrist_jog_minus_cbtn);
	command_button_cycle(hmi_wrist_phase_move_cbtn);
	command_button_cycle(hmi_wrist_copy_phase_cbtn);
	command_button_cycle(hmi_wrist_activate_pendant_cbtn);
	command_button_cycle(hmi_x_jog_plus_cbtn);
	command_button_cycle(hmi_x_jog_minus_cbtn);
	command_button_cycle(hmi_x_phase_move_cbtn);
	command_button_cycle(hmi_x_copy_phase_cbtn);
	command_button_cycle(hmi_x_activate_pendant_cbtn);
	command_button_cycle(hmi_y_jog_plus_cbtn);
	command_button_cycle(hmi_y_jog_minus_cbtn);
	command_button_cycle(hmi_y_phase_move_cbtn);
	command_button_cycle(hmi_y_copy_phase_cbtn);
	command_button_cycle(hmi_y_activate_pendant_cbtn);
	command_button_cycle(hmi_tilt_jog_plus_cbtn);
	command_button_cycle(hmi_tilt_jog_minus_cbtn);
	command_button_cycle(hmi_tilt_phase_move_cbtn);
	command_button_cycle(hmi_tilt_copy_phase_cbtn);
	command_button_cycle(hmi_tilt_activate_pendant_cbtn);
END_IF
END_ACTION

ACTION _read_process_image:
;
END_ACTION

ACTION _read_var_input:
;
END_ACTION

ACTION _set_runtime_properties:
elbow_actual_position			:= axis_get_actual_incremental_position(csp_case_feed_arm_elbow.axis);
shoulder_actual_position		:= axis_get_actual_incremental_position(csp_case_feed_arm_shoulder.axis);
wrist_actual_position			:= axis_get_actual_incremental_position(csp_case_feed_arm_wrist.axis);
x_actual_position				:= SEL(cartesian_mode_active, stAxesPosOut[1], axis_get_actual_incremental_position(csp_case_feed_kinematic_x.axis));
y_actual_position				:= SEL(cartesian_mode_active, stAxesPosOut[2], axis_get_actual_incremental_position(csp_case_feed_kinematic_y.axis));
tilt_actual_position			:= SEL(cartesian_mode_active, stAxesPosOut[3], axis_get_actual_incremental_position(csp_case_feed_kinematic_tilt.axis));

axis_are_moving :=
	axis_is_moving(csp_case_feed_arm_elbow.axis)
	OR
	axis_is_moving(csp_case_feed_arm_shoulder.axis)
	OR
	axis_is_moving(csp_case_feed_arm_wrist.axis)
	OR
	axis_is_moving(csp_case_feed_kinematic_x.axis)
	OR
	axis_is_moving(csp_case_feed_kinematic_y.axis)
	OR
	axis_is_moving(csp_case_feed_kinematic_tilt.axis);
	
visu_disable_general_command :=
	axis_are_moving
	OR 
	phase_request
	OR
	fbConfigKinGroup.bBusy
	OR
	motorization_manager_is_starting(csp_main_motorization_manager.motm)
	OR
	motorization_manager_is_execute(csp_main_motorization_manager.motm);	

visu_disable_ACS_command := 
	visu_disable_general_command
	OR
	kin_config_cartesian_mode;

visu_disable_MCS_command := 
	visu_disable_general_command
	OR
	NOT kin_config_cartesian_mode;
	
visu_disable_ACS_jog_mode :=
	kin_config_cartesian_mode 
	OR
	axis_are_phase_moving
	OR
	phase_request
	OR
	motorization_manager_is_starting(csp_main_motorization_manager.motm)
	OR
	motorization_manager_is_execute(csp_main_motorization_manager.motm);	

visu_disable_MCS_jog_mode :=
	NOT kin_config_cartesian_mode 
	OR
	axis_are_phase_moving
	OR
	phase_request
	OR
	motorization_manager_is_starting(csp_main_motorization_manager.motm)
	OR
	motorization_manager_is_execute(csp_main_motorization_manager.motm);	

visu_disable_phase_request := 
	axis_are_moving
	OR
	motorization_manager_is_starting(csp_main_motorization_manager.motm)
	OR
	motorization_manager_is_execute(csp_main_motorization_manager.motm);
END_ACTION

ACTION _write_output:
;
END_ACTION

END_PROGRAM

// ---- Application/CSP/Case/Feed/Kinematic/csp_case_feed_kinematic_x.TcPOU
	(*********************************** G.D S.p.A. - Technical Department ***********************************
============= PROGRAM INFO ============
FOLDER:             TBD
MACHINES INVOLVED:  TBD 

============= DESCRIPTION =============
csp machine declaration

============= REVISIONS ===============
Date		Version	 	Author      	Description             
----------	-------		------------  	--------------------------------------------
2019/04/05 	0000.00	 	M.Grasso		Creation of the PRG

**********************************************************************************************************)
(*$R process_ref := prc; $*)
PROGRAM csp_case_feed_kinematic_x
VAR
		
	prc:												process;
	prc_path:											STRING;
	
	axis:												axis;
	axis_actual_position:								LREAL;

	fsm_enable_condition:								BOOL := FALSE;
	fsm_next_status:									csp_case_feed_kinematic_status_enum;
	fsm_status:											csp_case_feed_kinematic_status_enum;
	debug_state_machine:								BOOL := FALSE;
	debug_state_machine_one_step:						BOOL := FALSE;	
	
	in_accu_safe_pos:                                   BOOL := FALSE;
    accu_tolerance:                                     LREAL := 5.0;
    accu_safe_pos:                                      LREAL := -745;
		
	cam_id:												INT := 2;
	
END_VAR

VAR CONSTANT
	(*Just in case you prefer having constants instead of numbers*)
	MOTOR_PHASE_VELOCITY_MMPS:							LREAL := 20;
	
	MOTOR_MAX_VELOCITY_MMPS:							LREAL := 1000;
	MOTOR_MAX_ACCELLERATION_MMPS2:						LREAL := 10000;
	MOTOR_MAX_DECELLERATION_MMPS2:						LREAL := 10000;
	MOTOR_MAX_JERK_MMPS3:								LREAL := 100000; 
	MOTOR_MAX_FOLLOWING_ERROR_MM:						LREAL := 10;
END_VAR

_read_var_input();

_object_manager();

IF NOT objects_running()
THEN
	RETURN;	
END_IF

_read_process_image();

_mode_manager();

CASE process_get_mode(prc) OF
	MODE_ABSENT,
	MODE_INACTIVE:
		RETURN;
	MODE_TEST:
		_handle_process_test();
END_CASE

_set_runtime_properties();

(********************************* BODY *********************************)

IF (axis.actual_position > (accu_safe_pos - accu_tolerance)) AND axis.actual_position < (accu_safe_pos + accu_tolerance)
THEN
	in_accu_safe_pos := TRUE;
ELSE
	in_accu_safe_pos := FALSE;   
END_IF

// Manage the accu change safe position
fsm_enable_condition := axis_is_ok(FALSE, axis)	
						AND															
						(csp_case_feed_kinematic.fsm_status = CSP_CASE_FEED_KINEMATIC_STATUS_ENABLED)
						AND
						csp_case_feed_kinematic.cartesian_mode_active
						AND							
						csp_main_accuChange.Brand_Change_Occurred;
										
IF	NOT fsm_enable_condition
	AND
	fsm_status <> CSP_CASE_FEED_KINEMATIC_STATUS_DISABLED	
THEN
	fsm_next_status	:= CSP_CASE_FEED_KINEMATIC_STATUS_DISABLED;
END_IF
					
CASE fsm_status OF
	
	CSP_CASE_FEED_KINEMATIC_STATUS_NOT_INITIALIZED:
	
        IF	axis_is_ok(return_when_absent := TRUE, CONVERSION_this := axis)
        THEN
            fsm_next_status := CSP_CASE_FEED_KINEMATIC_STATUS_DISABLED;
        END_IF

		
	CSP_CASE_FEED_KINEMATIC_STATUS_DISABLED:
	
		IF	fsm_enable_condition
			AND
			motorization_conditioner_is_execute(csp_main_services_towerLamp.buzzer_motcond) 							
		THEN	
			IF	in_accu_safe_pos
			THEN
				fsm_next_status := CSP_CASE_FEED_KINEMATIC_STATUS_CHANGE_OVER_MODE_DONE;
			ELSE								
				fsm_next_status := CSP_CASE_FEED_KINEMATIC_STATUS_ENABLED;
			END_IF
		END_IF;

		
	CSP_CASE_FEED_KINEMATIC_STATUS_ENABLED:	
	
		axis_move_absolute(
			position 		:= accu_safe_pos,
			velocity 		:= MOTOR_PHASE_VELOCITY_MMPS,
			direction		:= AXIS_CURRENT_DIRECTION,
			acceleration 	:= MOTOR_MAX_ACCELLERATION_MMPS2,
			deceleration 	:= MOTOR_MAX_DECELLERATION_MMPS2,
			jerk 			:= MOTOR_MAX_JERK_MMPS3, 
			buffer_mode 	:= AXIS_BUFFER_MODE_BUFFERED,
			CONVERSION_this := axis);
			
		IF 	axis_is_absolute_moving(axis)
		THEN
			fsm_next_status	:= CSP_CASE_FEED_KINEMATIC_STATUS_CHANGE_OVER_MODE;
		END_IF
		
		
	CSP_CASE_FEED_KINEMATIC_STATUS_CHANGE_OVER_MODE:
	
		IF 	axis_is_standstill(axis)
		THEN	
			axis_disable(axis);					
			fsm_next_status := CSP_CASE_FEED_KINEMATIC_STATUS_CHANGE_OVER_MODE_DONE;
		END_IF
		
		
	CSP_CASE_FEED_KINEMATIC_STATUS_CHANGE_OVER_MODE_DONE:
	
		;
		
END_CASE

IF 	NOT debug_state_machine
	OR
	debug_state_machine_one_step
THEN
	fsm_status := fsm_next_status;
	debug_state_machine_one_step := FALSE;
END_IF

(* TEMPORARY CAM CHANGE *)
IF csp_main_brand.count = '24Count'
	THEN
		cam_id := 302;
ELSIF csp_main_brand.count = '10Count'
	THEN
		cam_id := 571;
ELSIF csp_main_brand.count = '32Count'
	THEN
		cam_id := 2;
ELSIF csp_main_brand.count = '48Count'
	THEN
		cam_id := 38;
END_IF

(************************************************************************)

_handle_messages();

_write_output();

ACTION _handle_messages:
;
END_ACTION

ACTION _handle_process_test:
;
END_ACTION

ACTION _mode_manager:
IF process_mode_req_is_pending(prc)
THEN
    process_apply_mode_req_first_step(prc);
    CASE process_get_mode(prc) OF
        MODE_TO_ABSENT:
			;
        MODE_TO_INACTIVE:
			;
        MODE_TO_TEST:
			;
        MODE_TO_OPERATIONAL:
			;
    END_CASE
    process_apply_mode_req_second_step(prc);
END_IF
END_ACTION

ACTION _object_manager:
IF objects_initialization()
THEN
	sub_process_init(
		object_name					:= 'csp_case_feed_kinematic_x.prc', 
		process						:= csp_case_feed_kinematic.prc, 
		CONVERSION_this				:= prc);
		
	prc_path 						:= process_get_path(prc);
	
	axis_init(
		object_name					:= CONCAT(prc_path, '_axis'), 
		axis_type					:= AXIS_TYPE_VIRTUAL, 
		encoder_scaling_factor		:= G_VIRTUAL_ENCODER_SCALING_FACTOR_DEGPINC,
		modulo						:= G_NO_MODULO_DEG, 
		process						:= prc, 
		CONVERSION_this				:= axis);
	
	axis_set_max_dynamic(
		reference_velocity			:=	MOTOR_MAX_VELOCITY_MMPS,
		velocity					:=	MOTOR_MAX_VELOCITY_MMPS,
		acceleration				:=	MOTOR_MAX_ACCELLERATION_MMPS2,
		deceleration				:=	MOTOR_MAX_DECELLERATION_MMPS2,
		jerk						:=	MOTOR_MAX_JERK_MMPS3,
		following_error				:=	MOTOR_MAX_FOLLOWING_ERROR_MM,
		CONVERSION_this				:=	axis);
	
END_IF

IF objects_running()
THEN
	process_cycle(prc);
	axis_cycle(axis);

END_IF
END_ACTION

ACTION _read_process_image:
;
END_ACTION

ACTION _read_var_input:
;
END_ACTION

ACTION _set_runtime_properties:
axis_actual_position := axis_get_actual_incremental_position(axis);
END_ACTION

ACTION _write_output:
;
END_ACTION

END_PROGRAM

// ---- Application/CSP/Main/Services/Tower Lamp/csp_main_services_towerLamp.TcPOU
(********************* G.D S.p.A. - Technical Department *****************************

Date			Version		Author			Description             
----------      -------		-----------		----------------------------------------------
2015/12/23		0000.00		M.Grasso		Initial Release

DESCRIPTION:	

NOTES:        		 

**************************************************************************************)
(*$R process_ref := prc; $*)

PROGRAM csp_main_services_towerLamp
VAR
	prc:								process;
	prc_path:							STRING;
	
	tower_lamp:							signaling_device;
	
	blue_lamp:							lamp;
	green_lamp:							lamp;
	yellow_lamp:						lamp;
	red_lamp:							lamp;
	
	
    green_lt:                    	    BYTE := 1;
    blue_lt:                        	BYTE := 4;
    red_lt:                        		BYTE := 2;
   	yellow_lt:                        	BYTE := 3;
	
	
	
	buzzer_status_bool AT %Q*:			boolean;
	buzzer_lmp:							lamp;
	buzzer_volume AT %Q*: 				BYTE := 10; (*RANGE: 0-255, Buzzer Volume*)
	buzzer_do:							digital_output;
	buzzer_volume_des	: 				BYTE:=255;

	buzzer_motcond:						motorization_conditioner;
	buzzer_tmr:							timer;
	buzzer_time_ms:						INT:=1500;
	time_is_expired_rtrig:				R_TRIG;

	buzzer_req_bool_or:					boolean_or;
	
	buzzer_test_mode:					BOOL:=FALSE;
	
	TEST_signaling:						BOOL;

	count: 								INT := 0;
	buzzer_req_bool: 					BOOL;
	buzzer_filt: 						filter;
	buzzer_req_act: 					BOOL := FALSE;
	buzzer_req_act_old: 				BOOL := FALSE;
	Test_red_lt: 						BOOL := FALSE;
	Test_green_lt: 						BOOL := FALSE;
	Test_red_lt_flash: 					BOOL;
	
	
	(* REJECT PRESENT BUZZER VAR *)
	reject_present:						BOOL;
	reject_vol_up:						BOOL := TRUE;
	
	reject_rtrig:						R_trig;	
	Reject_Acknowledged: 				BOOL := FALSE; (*$P $*)
	
	reject_status_flt: 					filter;
	flt_timer_off_on: 					DINT := 10000; (*$P min := 0; max := 60000; step := 1; unit :=  ms; desc := Timer OFF to ON; $*)
	flt_timer_on_off: 					DINT := 200; (*$P min := 0; max := 10000; step := 1; unit :=  ms; desc := Timer ON to OFF; $*)
	
	reject_present_filtered: 			BOOL := FALSE;
	reject_ack_overwrite:				parameter_overwrite;
	
	Alarm_duration: TON;
	error_alarm_start: BOOL;
	error_alarm_complete: BOOL;

END_VAR

VAR_OUTPUT
	o_sim_buzzer_do_field_status:		BOOL;
	o_sim_blue_do_field_status:			BOOL;
	o_sim_green_field_status:			BOOL;
	o_sim_yellow_do_field_status:		BOOL;
	o_sim_red_do_field_status:			BOOL;
END_VAR

VAR_INPUT
	buzzer_request_ext: 				BOOL;
END_VAR

_read_var_input();
_sim_update();
_objects_manager();

IF g_application_status <> APPLICATION_STATUS_RUNNING
THEN
	RETURN;
END_IF

_read_process_image();

_mode_manager();

CASE process_get_mode (CONVERSION_this := prc) OF

	MODE_ABSENT,
	MODE_INACTIVE:
		//pwm_stop(FALSE, buzzer_pwm);
		RETURN;

	MODE_TEST:
		_handle_process_test();
END_CASE
_set_runtime_properties();

(*************************************************************************************
**************************************************************************************)
(* BODY *)

time_is_expired_rtrig(CLK := timer_is_expired(buzzer_tmr));

IF machine_has_message_typology_on(MESSAGE_TYPOLOGY_OBLIGATION , csp.mch) OR csp_case_feed_magazine_level.level_status> CSP_CASE_FEED_MAGAZINE_LEVEL_STATUS_LOW (*AMR 10012021*)
THEN
	tower_lamp.iol_slave_pdo_output.seg_2_color := blue_lt;
	lamp_on(blue_lamp);
ELSE
	tower_lamp.iol_slave_pdo_output.seg_2_color := 0;
	lamp_off(blue_lamp);
END_IF

IF machine_is_running(csp.mch) 
    OR
    machine_get_status(csp.mch)= MACHINE_STATUS_RUNNING
    OR
    Test_green_lt
THEN
    tower_lamp.iol_slave_pdo_output.seg_1_color := green_lt;
    
    ELSE
    tower_lamp.iol_slave_pdo_output.seg_1_color := 0;
END_IF

IF csp_main_motorization.held_BIT
OR csp_main_accuChange.accU_axis_moving
OR message_is_on(csp_case_discharge_reject_sensors.downstream_backup_di_dchk.alarm_asm.message)
THEN
    tower_lamp.iol_slave_pdo_output.seg_1_blink := TRUE;
    ELSE
    tower_lamp.iol_slave_pdo_output.seg_1_blink := FALSE;
END_IF

IF  machine_has_message_typology_on(MESSAGE_TYPOLOGY_ABNORMAL , csp.mch) 
    OR 
    machine_has_message_typology_on(MESSAGE_TYPOLOGY_EMERGENCY , csp.mch)
    OR
    machine_get_status(csp.mch)= MACHINE_STATUS_STOPPED
    OR 
    NOT machine_is_running(csp.mch)
    OR    
    Test_red_lt
	THEN
    tower_lamp.iol_slave_pdo_output.seg_3_color := red_lt;
    
ELSE
    tower_lamp.iol_slave_pdo_output.seg_3_color := 0;    
    
END_IF

IF machine_is_stop_emergency_active(csp.mch) 
    AND NOT machine_is_running(csp.mch)
    OR    
    Test_red_lt_flash
THEN
    tower_lamp.iol_slave_pdo_output.seg_3_blink := TRUE; 
    
ELSE
    tower_lamp.iol_slave_pdo_output.seg_3_blink := FALSE;    
    
END_IF

(*IF machine_is_stopping(csp.mch)
	AND NOT timer_is_expired(stop_timer)
	THEN
	
END_IF
*)

IF 	boolean_or_get_status(buzzer_req_bool_or)
	OR
	buzzer_test_mode
	OR
	machine_is_running_edge(csp.mch)
	OR
	buzzer_request_ext
		
THEN
	buzzer_req_bool := TRUE;
	buzzer_test_mode := FALSE;
	buzzer_request_ext := False;
ELSE
	buzzer_req_bool := FALSE;
END_IF

IF filter_is_on(buzzer_filt)
	THEN
		buzzer_req_act := TRUE;
	ELSE
		buzzer_req_act := FALSE;
END_IF

(* BUZZER HORN CONTROL ON/OFF *)
IF buzzer_req_act
OR (filter_is_on(reject_status_flt) AND machine_is_running(csp.mch) AND NOT Reject_Acknowledged)
OR filter_is_on(csp_main_accuchange.horn_on_filter)
OR error_alarm_start AND NOT error_alarm_complete
	THEN
		digital_output_set(buzzer_do);
ELSE
	digital_output_reset(buzzer_do);
END_IF


Alarm_duration(IN:= error_alarm_start , PT:=T#3S , Q=> error_alarm_complete , ET=> );

IF machine_is_stopped(csp.mch)
	THEN
	error_alarm_start := TRUE;
	ELSE
	error_alarm_start := FALSE;
END_IF

IF buzzer_req_act = FALSE AND buzzer_req_act_old = TRUE
	THEN
		motorization_conditioner_start_done(buzzer_motcond);
END_IF

buzzer_req_act_old := buzzer_req_act;

buzzer_volume := buzzer_volume_des;



(* REJECT PRESENT BUZZER LOGIC *)
IF message_is_on(csp_case_discharge_reject_sensors.reject_present_di_dchk.alarm_asm.message)
OR message_is_on(csp_transfer_crosspusher_reject.reject_present_check.alarm_asm.message)
OR message_is_on(csp_transfer_infeed_reject.bin_full_dchk.alarm_asm.message)
OR message_is_on(csp_case_discharge_reject_sensors.downstream_backup_di_dchk.alarm_asm.message)//added horn for discharge backup 
OR message_is_on(csp_case_feed_magazine_level_zonelow.magazine_level_zone_low_wem)
	THEN
		reject_present := TRUE;
ELSE
	reject_present := FALSE;
END_IF

IF reject_present
AND filter_is_off(reject_status_flt) 
	THEN
		reject_present_filtered := TRUE;
END_IF

IF filter_is_on(reject_status_flt)
	THEN
		reject_present_filtered := FALSE;
END_IF

filter_set_delays(
	delay_off_on			:= flt_timer_off_on,
	delay_on_off			:= flt_timer_on_off,
	CONVERSION_this			:= reject_status_flt);


reject_rtrig(clk := reject_present);

IF reject_rtrig.Q
	THEN
		parameter_overwrite_set_bool_value(FALSE, reject_ack_overwrite);
END_IF



(*IF TEST_signaling
    THEN
	    tower_lamp.iol_slave_pdo_output.seg_1_color := green_lt;
        tower_lamp.iol_slave_pdo_output.seg_2_color := red_lt;
        tower_lamp.iol_slave_pdo_output.seg_3_color := blue_lt;
       
